// TwinCAT 3 PLC project EngineeringToolbox
// Title: EngineeringToolbox
// Company: Beckhoff Electronics Mfg
// Author: Daniel Schlingmann
// ProjectVersion: 3.1.2.2
// Description: Engineering Toolbox Library The library is provided "as-is" for TwinCAT3.1 by the Beckhoff Industry Management for Electronics Manufacturing. Please check the function "DisclaimerStatement : WSTRING[1500]" in additon to the following disclaimer: THE SOFTWARE IS PROVIDED "AS IS", WITHOUT WARRANTY OF ANY KIND, EXPRESS OR IMPLIED, INCLUDING BUT NOT LIMITED TO THE WARRANTIES OF MERCHANTABILITY, FITNESS FOR A PARTICULAR PURPOSE AND NONINFRINGEMENT. IN NO EVENT SHALL THE AUTHORS OR COPYRIGHT HOLDERS BE LIABLE FOR ANY CLAIM, DAMAGES OR OTHER LIABILITY, WHETHER IN AN ACTION OF CONTRACT, TORT OR OTHERWISE, ARISING FROM, OUT OF OR IN CONNECTION WITH THE SOFTWARE OR THE USE OR OTHER DEALINGS IN THE SOFTWARE.
// ProgramVersion: 3.1.4022.7
// libraries:
//   Tc2_Drive, * (Beckhoff Automation GmbH)
//   Tc2_EtherCAT, * (Beckhoff Automation GmbH)
//   Tc2_IoFunctions, * (Beckhoff Automation GmbH)
//   Tc2_Math, * (Beckhoff Automation GmbH)
//   Tc2_MC2, * (Beckhoff Automation GmbH)
//   Tc2_MC2_Camming, * (Beckhoff Automation GmbH)
//   Tc2_MC2_Drive, * (Beckhoff Automation GmbH)
//   Tc2_MC2_FlyingSaw, * (Beckhoff Automation GmbH)
//   Tc2_MDP, * (Beckhoff Automation GmbH)
//   Tc2_ModbusRTU, * (Beckhoff Automation GmbH)
//   Tc2_ModbusSrv, * (Beckhoff Automation GmbH)
//   Tc2_NC, * (Beckhoff Automation GmbH)
//   Tc2_NCI, * (Beckhoff Automation GmbH)
//   Tc2_NcKinematicTransformation, * (Beckhoff Automation GmbH)
//   Tc2_PlcInterpolation, * (Beckhoff Automation GmbH)
//   Tc2_SerialCom, * (Beckhoff Automation GmbH)
//   Tc2_Smtp, * (Beckhoff Automation GmbH)
//   Tc2_Standard, * (Beckhoff Automation GmbH)
//   Tc2_SUPS, * (Beckhoff Automation GmbH)
//   Tc2_System, * (Beckhoff Automation GmbH)
//   Tc2_TcpIp, * (Beckhoff Automation GmbH)
//   Tc2_Utilities, * (Beckhoff Automation GmbH)
//   Tc2_XmlDataSrv, * (Beckhoff Automation GmbH)
//   Tc3_Module, * (Beckhoff Automation GmbH)
//   Tc2_BackupRestoreEL6900,newest,Beckhoff Automation GmbH
// project tree:
//   GVLs/ Gvl.TcGVL (not stored), PARAM.TcGVL (not stored)
//   POUs/BoundsCheck/ boundsError.TcPOU (not stored), boundsOK.TcPOU (not stored), checkBounds.TcPOU (not stored), CheckBoundsInfo.TcPOU (not stored)
//   POUs/Connectivity/ADS/ AdsDataExchange.TcPOU (not stored)
//   POUs/Connectivity/ Ipv4Addr_TO_UDINT.TcPOU (not stored), U_DEVICE_COM_CACHE.TcDUT, U_IPv4Addr.TcDUT (not stored), isValidIPv4Addr.TcPOU (not stored)
//   POUs/Connectivity/TF6310-TcpServer/DeviceCom/ TCPDeviceCom_SendRecBytes.TcPOU (not stored), TCPDeviceCom_SendRecString.TcPOU (not stored)
//   POUs/Connectivity/TF6340-SerialCom/ComPortDeviceCom/ ComPortDeviceCom_BufferHandle.TcPOU (not stored), ComPortDeviceCom_SendRecBytes.TcPOU (not stored), ComPortDeviceCom_SendRecString.TcPOU (not stored), ComPortEL6x22BEasyConnect.TcPOU (not stored)
//   POUs/Connectivity/TF6340-SerialCom/ComPortBasic/ ComPortBackground.TcPOU (not stored), ComPortSendRec.TcPOU (not stored)
//   POUs/Connectivity/TF625x-Modbus/Master/TF6250-ModbusTcpServer/TCP/ ModbusTcpMaster.TcPOU (not stored)
//   POUs/Connectivity/TF625x-Modbus/Master/TF6250-ModbusTcpServer/UDP/ ModbusUdpMaster.TcPOU (not stored)
//   POUs/Connectivity/TF625x-Modbus/Master/TF6255-ModbusRtu/ ModbusRtuMaster22B.TcPOU (not stored), ModbusRtuMaster5B.TcPOU (not stored), ModbusRtuMasterPC.TcPOU (not stored)
//   POUs/Connectivity/TF625x-Modbus/Master/_Components/ ModbusJob.TcPOU (not stored), ModbusSlaveCom.TcPOU (not stored)
//   POUs/Connectivity/TF625x-Modbus/Slave/ ModbusSlaveBase.TcPOU
//   POUs/Connectivity/TF6310-TcpServer/TcpBasic/ TCPSendRecCtrl.TcPOU (not stored), TCPConnectionCtrl.TcPOU (not stored), TCPSocketCtrl.TcPOU (not stored)
//   POUs/Connectivity/TF6310-TcpServer/UdpBasic/ UDPSendRecCtrl.TcPOU (not stored), UDPServerCtrl.TcPOU (not stored), UDPSocketCtrl.TcPOU (not stored)
//   POUs/ControllerTools/ AverageFilter.TcPOU, PIDController.TcPOU (not stored), PT1Filter.TcPOU (not stored), signum.TcPOU (not stored), SlewRateLimitter.TcPOU (not stored), SlidingAverageExt.TcPOU (not stored), SlidingAverage.TcPOU (not stored), ThreePointController.TcPOU (not stored)
//   POUs/DataBuffer/ DoubleBuffer.TcPOU (not stored), Quicksort.TcPOU (not stored)
//   POUs/DataBuffer/Fifo/ Fifo.TcPOU (not stored), FifoExt.TcPOU (not stored), FifoLRealSimple.TcPOU (not stored), FifoBase.TcPOU (not stored)
//   POUs/DataBuffer/Ringbuffer/ RingbufferBase.TcPOU (not stored), Ringbuffer.TcPOU (not stored), RingbufferCharSimple.TcPOU (not stored), RingbufferExt.TcPOU (not stored), RingbufferByteSimple.TcPOU (not stored), RingbufferLRealSimple.TcPOU (not stored)
//   POUs/EventLogger/ EventsWriteToLogbook.TcPOU (not stored), EVENT_HANDLING_CONFIG.TcDUT (not stored), getEventClassPriority.TcPOU (not stored), getEventClassText.TcPOU, SOURCE_ID.TcDUT (not stored)
//   POUs/EventLogger/ReadEvents/ EventlogRead.TcPOU (not stored), EVENTLOG_READ_DATA.TcDUT (not stored), EVENTLOG_READ_HANDLEINFO.TcDUT (not stored), EVENTLOG_READ_STREAM.TcDUT (not stored), EVENTLOG_READ_STREAM_DATA_RAW.TcDUT, EVENTLOG_READ_STREAM_DATA_RAW_EX.TcDUT (not stored)
//   POUs/EventLogger/TriggerEvents/ EventHandling.TcPOU (not stored), EventHandlingGrp10.TcPOU (not stored), EventHandlingGrp25.TcPOU (not stored), EventHandlingGrp50.TcPOU (not stored), EventHandlingGrpCustomized.TcPOU, EventHandlingConfirmIsReq.TcPOU, EventHandlingStatisticInfo.TcPOU (not stored)
//   POUs/Fieldbus/CANopen/ CANopenMasterDiag.TcPOU (not stored), CANopenMasterIO.TcPOU (not stored)
//   POUs/Fieldbus/EAP/ EAP_PUB_SUB_IO.TcPOU (not stored), EAP_DEVICE_IO.TcPOU (not stored), EAP_PUB_VAR.TcPOU (not stored), EAP_SUB_VAR.TcPOU (not stored)
//   POUs/Fieldbus/EtherCAT/ EcCoEReadNewestDiagMsg.TcPOU (not stored), EcDiagBase.TcPOU (not stored), EcDiagBase_wEvents.TcPOU (not stored)
//   POUs/Fieldbus/EtherCAT/_Components/ EcMasterIO.TcPOU (not stored), EcMasterSupervisor.TcPOU, EcSlavesDiag.TcPOU (not stored), EcSlaveSupervisor.TcPOU (not stored), EC_MASTER_DEVICE_STATE.TcDUT (not stored), EC_SLAVE_DIAG_INFO_DATA.TcDUT
//   POUs/Fieldbus/Profibus/ ProfibusMasterDiag.TcPOU (not stored), ProfibusMasterIO.TcPOU (not stored)
//   POUs/Fieldbus/Profinet/ ProfinetControllerIO.TcPOU, ProfinetControllerIO_wEvents.TcPOU (not stored), ProfinetDeviceIO.TcPOU (not stored)
//   POUs/FileHandling/Basic/ FileHandling.TcPOU (not stored), ReadDirSimple.TcPOU, ReadDirSimpleExt.TcPOU (not stored)
//   POUs/FileHandling/TF6421-XmlServer/ XmlReadWrite.TcPOU, XmlReadWriteWithBackupFile.TcPOU (not stored)
//   POUs/IO/Analog/ AnalogIn.TcPOU (not stored), AnalogIn32.TcPOU (not stored), AnalogInELMBase.TcPOU (not stored), AnalogInELMSingleSampleDINT.TcPOU (not stored), AnalogInELMSingleSampleREAL.TcPOU (not stored), AnalogInREAL.TcPOU (not stored), AnalogOut.TcPOU (not stored)
//   POUs/IO/ BlowOffSensors.TcPOU, Button.TcPOU (not stored), ButtonExt.TcPOU (not stored), Fuse.TcPOU (not stored), InOut.TcPOU (not stored), InOutExt.TcPOU (not stored), Input.TcPOU (not stored), Output.TcPOU
//   POUs/IO/Cylinder/ Cylinder.TcPOU (not stored), CylinderExt.TcPOU, CylinderType4.TcPOU (not stored), I_Cylinder.TcIO (not stored)
//   POUs/IO/Drives/ AxDriveBase.TcPOU, AxDriveGetRef.TcPOU (not stored), I_AxDriveBase.TcIO (not stored)
//   POUs/IO/Drives/CoE/ AxDriveCoE.TcPOU (not stored), AxDriveCoE_wEvents.TcPOU (not stored), CiA_DS402Controlword.TcPOU, CiA_DS402Statusword.TcPOU (not stored), eCiA_DS402_CONTROL_CMD.TcDUT (not stored), eCiA_DS402_STATUS_STATE.TcDUT (not stored)
//   POUs/IO/Drives/CoE/EL72xx/ AxDriveCoE_EL72xxParam.TcPOU (not stored), CiA_DS402StatuswordEx7xxx.TcPOU (not stored)
//   POUs/IO/Drives/DC/Ey73xx/ AxDriveDC.TcPOU, AxDriveDC_wEvents.TcPOU (not stored)
//   POUs/IO/Drives/SoE/ AxDriveSoE_Ax5000CommutationCalib.TcPOU (not stored), AxDriveSoE_Ax5000CalcPower.TcPOU (not stored), AxDriveSoE_Ax5000SwitchParamSet.TcPOU (not stored), Ax580x.TcPOU (not stored), AxDriveSoE_Ax5000.TcPOU (not stored), AxDriveSoE_Ax5000Param.TcPOU (not stored), AxDriveSoE_Ax5000wEvents.TcPOU (not stored), AxDriveSoE_Rexroth.TcPOU
//   POUs/IO/Drives/SoE/Ax5000ParamSTRUCTs/P/ AX5000_P_0001.TcDUT (not stored), AX5000_P_0002.TcDUT (not stored), AX5000_P_0003.TcDUT (not stored), AX5000_P_0004.TcDUT (not stored), AX5000_P_0009.TcDUT (not stored), AX5000_P_0010.TcDUT (not stored), AX5000_P_0020.TcDUT (not stored), AX5000_P_0021.TcDUT (not stored), AX5000_P_0040.TcDUT (not stored), AX5000_P_0050.TcDUT (not stored), AX5000_P_0051.TcDUT (not stored), AX5000_P_0052.TcDUT, AX5000_P_0053.TcDUT (not stored), AX5000_P_0054.TcDUT (not stored), AX5000_P_0055.TcDUT (not stored), AX5000_P_0056.TcDUT (not stored), AX5000_P_0057.TcDUT (not stored), AX5000_P_0058.TcDUT (not stored), AX5000_P_0059.TcDUT (not stored), AX5000_P_0060.TcDUT (not stored), AX5000_P_0061.TcDUT (not stored), AX5000_P_0062.TcDUT (not stored), AX5000_P_0063.TcDUT (not stored), AX5000_P_0064.TcDUT (not stored), AX5000_P_0065.TcDUT (not stored), AX5000_P_0066.TcDUT (not stored), AX5000_P_0067.TcDUT (not stored), AX5000_P_0068.TcDUT (not stored), AX5000_P_0069.TcDUT (not stored), AX5000_P_0070.TcDUT (not stored), AX5000_P_0071.TcDUT (not stored), AX5000_P_0072.TcDUT (not stored), AX5000_P_0073.TcDUT, AX5000_P_0074.TcDUT (not stored), AX5000_P_0075.TcDUT (not stored), AX5000_P_0076.TcDUT (not stored), AX5000_P_0077.TcDUT (not stored), AX5000_P_0078.TcDUT (not stored), AX5000_P_0088.TcDUT (not stored), AX5000_P_0089.TcDUT (not stored), AX5000_P_0090.TcDUT (not stored), AX5000_P_0091.TcDUT (not stored), AX5000_P_0092.TcDUT, AX5000_P_0093.TcDUT (not stored), AX5000_P_0096.TcDUT (not stored), AX5000_P_0097.TcDUT (not stored), AX5000_P_0098_beckhoff.TcDUT (not stored), AX5000_P_0098_beckhoff_electrical_data.TcDUT (not stored), AX5000_P_0099.TcDUT (not stored), AX5000_P_0100.TcDUT (not stored), AX5000_P_0101.TcDUT (not stored), AX5000_P_0102.TcDUT (not stored), AX5000_P_0103.TcDUT (not stored), AX5000_P_0104.TcDUT (not stored), AX5000_P_0105.TcDUT (not stored), AX5000_P_0106.TcDUT (not stored), AX5000_P_0107.TcDUT (not stored), AX5000_P_0108.TcDUT (not stored), AX5000_P_0109.TcDUT (not stored), AX5000_P_0110.TcDUT (not stored), AX5000_P_0111.TcDUT (not stored), AX5000_P_0112.TcDUT (not stored), AX5000_P_0113.TcDUT (not stored), AX5000_P_0114.TcDUT (not stored), AX5000_P_0115.TcDUT (not stored), AX5000_P_0116.TcDUT (not stored), AX5000_P_0117.TcDUT (not stored), AX5000_P_0118.TcDUT (not stored), AX5000_P_0119.TcDUT (not stored), AX5000_P_0125.TcDUT (not stored), AX5000_P_0126.TcDUT, AX5000_P_0127.TcDUT (not stored), AX5000_P_0128.TcDUT, AX5000_P_0150.TcDUT, AX5000_P_0151.TcDUT (not stored), AX5000_P_0152.TcDUT (not stored), AX5000_P_0153.TcDUT (not stored), AX5000_P_0154.TcDUT (not stored), AX5000_P_0155.TcDUT (not stored), AX5000_P_0158.TcDUT (not stored), AX5000_P_0159.TcDUT (not stored), AX5000_P_0160.TcDUT, AX5000_P_0161.TcDUT (not stored), AX5000_P_0162.TcDUT (not stored), AX5000_P_0163.TcDUT, AX5000_P_0165.TcDUT (not stored), AX5000_P_0166.TcDUT (not stored), AX5000_P_0167.TcDUT (not stored), AX5000_P_0168.TcDUT (not stored), AX5000_P_0169.TcDUT (not stored), AX5000_P_0170.TcDUT (not stored), AX5000_P_0171.TcDUT (not stored), AX5000_P_0180.TcDUT, AX5000_P_0181.TcDUT (not stored), AX5000_P_0182.TcDUT (not stored), AX5000_P_0183.TcDUT, AX5000_P_0184.TcDUT (not stored), AX5000_P_0185.TcDUT (not stored), AX5000_P_0188.TcDUT (not stored), AX5000_P_0189.TcDUT (not stored), AX5000_P_0192.TcDUT (not stored), AX5000_P_0193.TcDUT (not stored), AX5000_P_0196.TcDUT (not stored), AX5000_P_0198.TcDUT (not stored), AX5000_P_0199.TcDUT (not stored), AX5000_P_0200.TcDUT (not stored), AX5000_P_0201.TcDUT, AX5000_P_0202.TcDUT (not stored), AX5000_P_0203.TcDUT (not stored), AX5000_P_0204.TcDUT (not stored), AX5000_P_0205.TcDUT (not stored), AX5000_P_0206.TcDUT (not stored), AX5000_P_0207.TcDUT (not stored), AX5000_P_0208.TcDUT (not stored), AX5000_P_0209.TcDUT (not stored), AX5000_P_0210.TcDUT, AX5000_P_0211.TcDUT (not stored), AX5000_P_0212.TcDUT (not stored), AX5000_P_0213.TcDUT (not stored), AX5000_P_0214.TcDUT, AX5000_P_0215.TcDUT (not stored), AX5000_P_0216.TcDUT (not stored), AX5000_P_0217.TcDUT (not stored), AX5000_P_0218.TcDUT (not stored), AX5000_P_0219.TcDUT (not stored), AX5000_P_0220.TcDUT (not stored), AX5000_P_0221.TcDUT (not stored), AX5000_P_0250.TcDUT (not stored), AX5000_P_0251.TcDUT (not stored), AX5000_P_0252.TcDUT (not stored), AX5000_P_0253.TcDUT (not stored), AX5000_P_0254.TcDUT (not stored), AX5000_P_0255.TcDUT (not stored), AX5000_P_0256.TcDUT (not stored), AX5000_P_0270.TcDUT, AX5000_P_0271.TcDUT (not stored), AX5000_P_0272.TcDUT (not stored), AX5000_P_0273.TcDUT (not stored), AX5000_P_0274.TcDUT, AX5000_P_0275.TcDUT (not stored), AX5000_P_0276.TcDUT, AX5000_P_0277.TcDUT (not stored), AX5000_P_0278.TcDUT (not stored), AX5000_P_0300.TcDUT (not stored), AX5000_P_0301.TcDUT (not stored), AX5000_P_0302.TcDUT (not stored), AX5000_P_0303.TcDUT (not stored), AX5000_P_0304.TcDUT (not stored), AX5000_P_0305.TcDUT (not stored), AX5000_P_0306.TcDUT (not stored), AX5000_P_0307.TcDUT (not stored), AX5000_P_0308.TcDUT (not stored), AX5000_P_0309.TcDUT (not stored), AX5000_P_0310.TcDUT (not stored), AX5000_P_0311.TcDUT, AX5000_P_0312.TcDUT (not stored), AX5000_P_0313.TcDUT, AX5000_P_0314.TcDUT (not stored), AX5000_P_0315.TcDUT (not stored), AX5000_P_0316.TcDUT (not stored), AX5000_P_0317.TcDUT (not stored), AX5000_P_0320.TcDUT (not stored), AX5000_P_0321.TcDUT (not stored), AX5000_P_0322.TcDUT (not stored), AX5000_P_0323.TcDUT (not stored), AX5000_P_0324.TcDUT, AX5000_P_0325.TcDUT, AX5000_P_0326.TcDUT (not stored), AX5000_P_0350.TcDUT (not stored), AX5000_P_0351.TcDUT (not stored), AX5000_P_0352.TcDUT (not stored), AX5000_P_0353.TcDUT (not stored), AX5000_P_0354.TcDUT (not stored), AX5000_P_0356.TcDUT (not stored), AX5000_P_0360.TcDUT (not stored), AX5000_P_0361.TcDUT (not stored), AX5000_P_0400.TcDUT (not stored), AX5000_P_0401.TcDUT (not stored), AX5000_P_0402.TcDUT (not stored), AX5000_P_0451.TcDUT (not stored), AX5000_P_0452.TcDUT (not stored), AX5000_P_0453.TcDUT (not stored), AX5000_P_0454.TcDUT (not stored), AX5000_P_0455.TcDUT (not stored), AX5000_P_0456.TcDUT, AX5000_P_0457.TcDUT (not stored), AX5000_P_0458.TcDUT (not stored), AX5000_P_0459.TcDUT (not stored), AX5000_P_0460.TcDUT (not stored), AX5000_P_0461.TcDUT (not stored), AX5000_P_0462.TcDUT (not stored), AX5000_P_0463.TcDUT (not stored), AX5000_P_0464.TcDUT (not stored), AX5000_P_0502.TcDUT (not stored), AX5000_P_0503.TcDUT (not stored), AX5000_P_0504.TcDUT (not stored), AX5000_P_0505.TcDUT (not stored), AX5000_P_0511.TcDUT (not stored), AX5000_P_0512.TcDUT (not stored), AX5000_P_0513.TcDUT (not stored), AX5000_P_0514.TcDUT (not stored), AX5000_P_0515.TcDUT (not stored), AX5000_P_0516.TcDUT (not stored), AX5000_P_0517.TcDUT (not stored), AX5000_P_0518.TcDUT (not stored), AX5000_P_0552.TcDUT (not stored), AX5000_P_0553.TcDUT (not stored), AX5000_P_0554.TcDUT (not stored), AX5000_P_0555.TcDUT (not stored), AX5000_P_0556.TcDUT, AX5000_P_0557.TcDUT (not stored), AX5000_P_0558.TcDUT (not stored), AX5000_P_0601.TcDUT (not stored), AX5000_P_0602.TcDUT, AX5000_P_0610.TcDUT, AX5000_P_0611.TcDUT (not stored), AX5000_P_0800.TcDUT (not stored), AX5000_P_0801.TcDUT (not stored), AX5000_P_0802.TcDUT (not stored), AX5000_P_0804.TcDUT, AX5000_P_0805.TcDUT (not stored), AX5000_P_0806.TcDUT (not stored), AX5000_P_0810.TcDUT (not stored), AX5000_P_0811.TcDUT (not stored), AX5000_P_0850.TcDUT (not stored), AX5000_P_0851.TcDUT (not stored), AX5000_P_0900.TcDUT (not stored), AX5000_P_0901.TcDUT (not stored), AX5000_P_0902.TcDUT (not stored), AX5000_P_0904.TcDUT (not stored), AX5000_P_0905.TcDUT, AX5000_P_0906.TcDUT (not stored), AX5000_P_0912.TcDUT (not stored), AX5000_P_1000.TcDUT, AX5000_P_1001.TcDUT (not stored), AX5000_P_1002.TcDUT (not stored), AX5000_P_1003.TcDUT (not stored), AX5000_P_1004.TcDUT, AX5000_P_1005.TcDUT (not stored), AX5000_P_1006.TcDUT (not stored), AX5000_P_1007.TcDUT (not stored), AX5000_P_1008.TcDUT (not stored), AX5000_P_1009.TcDUT (not stored), AX5000_P_1010.TcDUT (not stored), AX5000_P_1011.TcDUT (not stored), AX5000_P_1012.TcDUT (not stored), AX5000_P_1020.TcDUT (not stored), AX5000_P_1021.TcDUT (not stored), AX5000_P_1022.TcDUT (not stored), AX5000_P_2000.TcDUT (not stored), AX5000_P_2001.TcDUT (not stored), AX5000_P_2002.TcDUT (not stored)
//   POUs/IO/Drives/SoE/Ax5000ParamSTRUCTs/S/ AX5000_S_0001.TcDUT (not stored), AX5000_S_0002.TcDUT (not stored), AX5000_S_0007.TcDUT, AX5000_S_0011.TcDUT (not stored), AX5000_S_0012.TcDUT (not stored), AX5000_S_0013.TcDUT (not stored), AX5000_S_0015.TcDUT (not stored), AX5000_S_0016.TcDUT (not stored), AX5000_S_0017.TcDUT (not stored), AX5000_S_0018.TcDUT (not stored), AX5000_S_0024.TcDUT (not stored), AX5000_S_0029.TcDUT (not stored), AX5000_S_0030.TcDUT (not stored), AX5000_S_0031.TcDUT (not stored), AX5000_S_0032.TcDUT (not stored), AX5000_S_0033.TcDUT (not stored), AX5000_S_0034.TcDUT (not stored), AX5000_S_0035.TcDUT (not stored), AX5000_S_0036.TcDUT (not stored), AX5000_S_0037.TcDUT (not stored), AX5000_S_0040.TcDUT (not stored), AX5000_S_0043.TcDUT (not stored), AX5000_S_0044.TcDUT (not stored), AX5000_S_0045.TcDUT (not stored), AX5000_S_0046.TcDUT (not stored), AX5000_S_0047.TcDUT (not stored), AX5000_S_0048.TcDUT (not stored), AX5000_S_0051.TcDUT, AX5000_S_0053.TcDUT (not stored), AX5000_S_0055.TcDUT (not stored), AX5000_S_0076.TcDUT, AX5000_S_0079.TcDUT (not stored), AX5000_S_0080.TcDUT (not stored), AX5000_S_0081.TcDUT (not stored), AX5000_S_0082.TcDUT (not stored), AX5000_S_0083.TcDUT (not stored), AX5000_S_0084.TcDUT (not stored), AX5000_S_0085.TcDUT (not stored), AX5000_S_0086.TcDUT (not stored), AX5000_S_0091.TcDUT (not stored), AX5000_S_0092.TcDUT (not stored), AX5000_S_0095.TcDUT (not stored), AX5000_S_0099.TcDUT (not stored), AX5000_S_0100.TcDUT (not stored), AX5000_S_0101.TcDUT, AX5000_S_0103.TcDUT (not stored), AX5000_S_0104.TcDUT (not stored), AX5000_S_0106.TcDUT (not stored), AX5000_S_0107.TcDUT (not stored), AX5000_S_0109.TcDUT, AX5000_S_0110.TcDUT, AX5000_S_0111.TcDUT (not stored), AX5000_S_0112.TcDUT (not stored), AX5000_S_0113.TcDUT (not stored), AX5000_S_0119.TcDUT (not stored), AX5000_S_0120.TcDUT, AX5000_S_0124.TcDUT (not stored), AX5000_S_0126.TcDUT (not stored), AX5000_S_0130.TcDUT (not stored), AX5000_S_0131.TcDUT (not stored), AX5000_S_0134.TcDUT (not stored), AX5000_S_0135.TcDUT, AX5000_S_0136.TcDUT, AX5000_S_0137.TcDUT, AX5000_S_0143.TcDUT (not stored), AX5000_S_0149.TcDUT (not stored), AX5000_S_0159.TcDUT (not stored), AX5000_S_0160.TcDUT (not stored), AX5000_S_0161.TcDUT (not stored), AX5000_S_0162.TcDUT (not stored), AX5000_S_0163.TcDUT (not stored), AX5000_S_0169.TcDUT (not stored), AX5000_S_0170.TcDUT (not stored), AX5000_S_0179.TcDUT (not stored), AX5000_S_0185.TcDUT (not stored), AX5000_S_0186.TcDUT (not stored), AX5000_S_0187.TcDUT (not stored), AX5000_S_0188.TcDUT (not stored), AX5000_S_0189.TcDUT (not stored), AX5000_S_0196.TcDUT (not stored), AX5000_S_0200.TcDUT (not stored), AX5000_S_0201.TcDUT, AX5000_S_0203.TcDUT (not stored), AX5000_S_0204.TcDUT (not stored), AX5000_S_0206.TcDUT (not stored), AX5000_S_0207.TcDUT (not stored), AX5000_S_0216.TcDUT (not stored), AX5000_S_0217.TcDUT (not stored), AX5000_S_0219.TcDUT (not stored), AX5000_S_0254.TcDUT (not stored), AX5000_S_0256.TcDUT (not stored), AX5000_S_0257.TcDUT (not stored), AX5000_S_0267.TcDUT (not stored), AX5000_S_0273.TcDUT (not stored), AX5000_S_0274.TcDUT (not stored), AX5000_S_0292.TcDUT (not stored), AX5000_S_0295.TcDUT (not stored), AX5000_S_0296.TcDUT, AX5000_S_0347.TcDUT (not stored), AX5000_S_0348.TcDUT (not stored), AX5000_S_0372.TcDUT (not stored), AX5000_S_0374.TcDUT, AX5000_S_0375.TcDUT (not stored), AX5000_S_0380.TcDUT (not stored), AX5000_S_0381.TcDUT (not stored), AX5000_S_0383.TcDUT (not stored), AX5000_S_0384.TcDUT (not stored), AX5000_S_0390.TcDUT, AX5000_S_0403.TcDUT (not stored), AX5000_S_0405.TcDUT (not stored), AX5000_S_0409.TcDUT, AX5000_S_0410.TcDUT (not stored), AX5000_S_0429.TcDUT (not stored), AX5000_S_0432.TcDUT (not stored), AX5000_S_0435.TcDUT (not stored), AX5000_S_0436.TcDUT (not stored)
//   POUs/IO/Drives/Stepper/ AxDriveStepper.TcPOU (not stored), AxDriveStepperParam.TcPOU, AxDriveStepper_wEvents.TcPOU (not stored)
//   POUs/IO/EL-EP/ AnalogOut_EL2535.TcPOU (not stored), EL1262_Base.TcPOU (not stored), EL3681.TcPOU (not stored), EL1904.TcPOU (not stored), EL69xx.TcPOU (not stored), EL3356.TcPOU (not stored), Eyx9xx.TcPOU (not stored), ZB8610.TcPOU (not stored)
//   POUs/IO/EL-EP/EL9x/ EL9501.TcPOU (not stored), EL9576.TcPOU, EL95xxPowerTerminal.TcPOU (not stored), ELSystemTerminal.TcPOU (not stored)
//   POUs/IO/_EcSlaveFWUpdater/ EcSlaveDevFWUpdater.TcPOU (not stored)
//   POUs/IO/_EcSlaveInfoDataIO/ EcSlaveInfoData.TcPOU (not stored), EcSlaveInfoDataExt.TcPOU (not stored), I_EcSlaveInfoData.TcIO (not stored)
//   POUs/IO/EL-EP/EL3403/ EL3403.TcPOU (not stored), EL3403Logic.TcPOU (not stored)
//   POUs/IO/EL-EP/EP92xxPwrBox/ EP9214.TcPOU (not stored), EP9214_CHANNEL.TcPOU (not stored), EP9224_0037.TcPOU (not stored), EP9224_0037_CHANNEL.TcPOU (not stored)
//   POUs/IO/FreqConv/EtherCAT/DS402/ EcFcDS402_ComBase.TcPOU
//   POUs/IO/FreqConv/ IOFcCom.TcPOU
//   POUs/IO/Motors/ IOMotor.TcPOU (not stored), IOMotor2Dir.TcPOU (not stored), IOMotorStarDelta.TcPOU (not stored)
//   POUs/IO/[underDev]/ Cylinder_wUnitItf.TcPOU (not stored)
//   POUs/IO/_ItfActuators/ I_ActuatorBase.TcIO (not stored), I_ActuatorEnableDisable.TcIO (not stored), I_ActuatorFwdRev.TcIO (not stored), I_ActuatorFwdBwd.TcIO (not stored), I_ActuatorLeftRight.TcIO (not stored), I_ActuatorOnOff.TcIO, I_ActuatorOpenClose.TcIO (not stored), I_ActuatorPosNeg.TcIO (not stored), I_ActuatorStartStop.TcIO (not stored), I_ActuatorUpDown.TcIO (not stored), I_ActuatorWorkBase.TcIO (not stored)
//   POUs/IpcDiag/MDP/InfoModuls/ MDP_CPU.TcPOU (not stored), MDP_Fan.TcPOU (not stored), MDP_Mainboard.TcPOU (not stored), MDP_RaidSimple.TcPOU (not stored), MDP_ReadModulList.TcPOU (not stored), MDP_SiliconDrives.TcPOU (not stored), MDP_UPS.TcPOU (not stored)
//   POUs/IpcDiag/MDP/ MDP_Info.TcPOU (not stored), MDP_IpcDiag.TcPOU (not stored), MDP_IpcDiag_wEvents.TcPOU (not stored)
//   POUs/IpcDiag/ UPSStatus.TcPOU (not stored)
//   POUs/Logging/ DataFileLogger.TcPOU (not stored), DataUdpLogger.TcPOU (not stored), I_LogbookSubscriber.TcIO (not stored), I_Logbook.TcIO (not stored), Logbook.TcPOU (not stored), LogbookData.TcDUT (not stored), LogbookPuplisher.TcPOU (not stored), LogbookSubEventLog.TcPOU, LogbookSubSendMail.TcPOU (not stored), adsLogError.TcPOU (not stored), adsLogHint.TcPOU (not stored), adsLogWarn.TcPOU (not stored), LogbookSubSysLog.TcPOU (not stored), LogbookSubWriteFile.TcPOU (not stored), Logbook_wEventClass.TcPOU (not stored), adsLogwTcEventClass.TcPOU (not stored)
//   POUs/Motion/TF50xx-NC/00_Base/ I_AxNcPTP.TcIO (not stored), AxFbBase.TcPOU (not stored), AxRWParaBase.TcPOU, I_AxNcBase.TcIO (not stored)
//   POUs/Motion/TF50xx-NC/02_Options/Parameter/ AxPara.TcPOU (not stored), AxParaCtrl.TcPOU (not stored)
//   POUs/Motion/TF50xx-NC/03_Utilities/ AxAutoWriteSoftLimit.TcPOU (not stored), CoordinateTransformation2D.TcPOU (not stored), AxCalcPosBias.TcPOU (not stored), AxResonanceAvoidance.TcPOU (not stored) (excluded from build), AxSoftSyncDistance.TcPOU, AxStatemodel.TcPOU (not stored), AxAutoFct.TcPOU (not stored), AX_JOB.TcPOU (not stored), getOvrVelo.TcPOU (not stored)
//   POUs/Motion/TF50xx-NC/ AxNcPTPwJobs.TcPOU (not stored), AxNcBaseExt.TcPOU (not stored), AxNcPtpGear.TcPOU (not stored), AxNcBase.TcPOU (not stored), AxNcPTP.TcPOU (not stored)
//   POUs/Motion/TF5100-NCI/ NciChannel_wEvents.TcPOU (not stored), NciChannel.TcPOU (not stored)
//   POUs/Motion/TF511x-KIN/03_DUTs/Positions/ KIN_POSITIONS.TcPOU (not stored), KIN_POSITIONS_ACS_DUT.TcDUT (not stored), KIN_POSITIONS_MCS_DUT.TcDUT (not stored), U_KIN_POSITIONS.TcDUT (not stored)
//   POUs/Motion/TF511x-KIN/03_DUTs/Trafo/ KIN_CALCTRAFO_AXPOS_PARAM.TcPOU (not stored), KIN_STATE_OBSERVER_OID_PARAM.TcPOU (not stored), KIN_STATICTRAFO_PARAM.TcPOU (not stored), KIN_TOOLTRAFO_PARAM.TcPOU (not stored), UCS.TcPOU (not stored)
//   POUs/Motion/ VALUE_3D.TcPOU (not stored), VALUE_3D_DUT.TcDUT (not stored), VALUE_6D.TcPOU, VALUE_6D_DUT.TcDUT (not stored)
//   POUs/Safety/Diag/ SafetyLogicAndIOTerminalDiag.TcPOU (not stored), SafetyIODeviceDiagRead.TcPOU (not stored), SafetyIODeviceDiag_wEvents.TcPOU (not stored), SafetyIOsDiag.TcPOU (not stored), SafetyLogicTerminalDiag.TcPOU (not stored), SafetyPlcTerminalDiag.TcPOU (not stored)
//   POUs/StringHelper/ cutStrNumberToSeperator.TcPOU (not stored), cutStrToSeperator2.TcPOU (not stored), replaceUmlauts.TcPOU (not stored), cutStrToSeperator.TcPOU, cutWStrToSeperator.TcPOU (not stored), DWORD_TO_BINSTR_EXT.TcPOU (not stored), DWORD_TO_HEXSTR_EXT.TcPOU, getCntCharInStr.TcPOU (not stored), getCntCharInWStr.TcPOU (not stored), isWStringNumeric.TcPOU (not stored), HEXSTR_TO_DWORD.TcPOU (not stored), HEXSTR_TO_LWORD.TcPOU (not stored), INSERT_EXT.TcPOU (not stored), LWORD_TO_BINSTR_EXT.TcPOU (not stored), LWORD_TO_HEXSTR_EXT.TcPOU (not stored), readStrToSeperator.TcPOU (not stored), replaceInString.TcPOU (not stored), getFilledString.TcPOU (not stored), isStringNumeric.TcPOU (not stored), readWStrToSeperator.TcPOU (not stored), replaceInWString.TcPOU (not stored), U_MAX_STRING.TcDUT (not stored), U_MAX_WSTRING.TcDUT (not stored), WINSERT_EXT.TcPOU (not stored)
//   POUs/System/ SystemInfo.TcPOU (not stored), SystemInfo64.TcPOU (not stored) (excluded from build), SystemPulses.TcPOU (not stored), TaskInfo.TcPOU (not stored)
//   POUs/TimeHelper/ PartsPerTime.TcPOU (not stored), createTOD.TcPOU (not stored), getDateAndTimeDelta.TcPOU (not stored), getTonCountdown.TcPOU (not stored), LivebitCheck.TcPOU (not stored), Ontime.TcPOU (not stored), OntimeExt.TcPOU (not stored), OntimeSimple.TcPOU (not stored), Pulse.TcPOU, SensorTimeoutCheck.TcPOU (not stored), systemtimeInCam.TcPOU (not stored), systemtimeCmp.TcPOU (not stored), systemtimeInWin.TcPOU (not stored), TimeSwitch.TcPOU (not stored), TONRecord.TcPOU (not stored), TONTOF.TcPOU (not stored), VeloLinearMeasurement.TcPOU (not stored)
//   POUs/_Miscellaneous/64BitFunctions/ CLEARBIT64.TcPOU (not stored), CSETBIT64.TcPOU (not stored), GETBIT64.TcPOU (not stored), SETBIT64.TcPOU (not stored)
//   POUs/_Miscellaneous/ nextIdx.TcPOU (not stored), TC_VN_COLORS.TcDUT (not stored) (excluded from build), FbBase.TcPOU (not stored), CAM.TcPOU, CAM3D.TcPOU (not stored), COLOR.TcDUT (not stored), ERROR_HDL.TcPOU (not stored), FbBaseExt.TcPOU (not stored), FbBaseOutputs.TcPOU (not stored), getNoOfBits.TcPOU, LCID.TcDUT (not stored), eLCID.TcDUT (not stored), LOGx.TcPOU (not stored), OEECalculation.TcPOU (not stored), polynomial.TcPOU (not stored), RF_TRIG.TcPOU (not stored), scale.TcPOU (not stored), SEQUENCE_HDL.TcPOU (not stored), setNoOfBits.TcPOU, TEST_FB.TcPOU (not stored), TOGGLE.TcPOU (not stored), U_32BIT_DATATYPE.TcDUT (not stored), U_64BIT_DATATYPE.TcDUT (not stored), WIN.TcPOU (not stored)
//   POUs/_Miscellaneous/Conversions/ ADSERROR_TO_HRESULT.TcPOU (not stored), DWORD_TO_REAL_EX.TcPOU (not stored), HRESULT_TO_ADSERROR.TcPOU (not stored), REAL_TO_FMLREAL.TcPOU (not stored), LWORD_TO_LREAL_EX.TcPOU (not stored), SWAP_BYTES_OF_WORDS.TcPOU (not stored), SWAP_WORDS_OF_DWORD.TcPOU (not stored), SWAP_WORDS_OF_LWORD.TcPOU (not stored), ADSERROR_TO_WIN32ERROR.TcPOU, ADSERROR_TO_WSERROR.TcPOU (not stored), C_TO_F.TcPOU (not stored), DEGREES_TO_RPM.TcPOU (not stored), F_TO_C.TcPOU (not stored), GF_TO_N.TcPOU (not stored), TO_FMLREAL.TcPOU (not stored), MMIN_TO_MMS.TcPOU, MMS_TO_MMIN.TcPOU, N_TO_GF.TcPOU (not stored), RPM_TO_DEGREES.TcPOU (not stored)
//   POUs/Safety/ SafetyCircuit.TcPOU (not stored), SafetyGroupIO.TcPOU (not stored), SafetyPlcBackupRestore.TcPOU (not stored), SAFETY_CIRCUIT_STATUS.TcDUT (not stored)
//   POUs/Statemodel/control/ I_StatemodelBase.TcIO (not stored), I_Statemodel.TcIO, Statemodel.TcPOU (not stored)
//   POUs/Statemodel/ eMODE.TcDUT, eSTATE.TcDUT (not stored)
//   POUs/Statemodel/UnitTemplate/ I_Statemodel_Unit.TcIO (not stored), Statemodel_Unit.TcPOU (not stored)
//   POUs/Motion/TF50xx-NC/01_Main/ AxAdmin.TcPOU (not stored), AxHoming.TcPOU, AxMotion.TcPOU (not stored)
//   POUs/Motion/TF50xx-NC/02_Options/Motion/ AxSuperposition.TcPOU (not stored), AxMoveSinus.TcPOU (not stored), AxHomingOnBlock.TcPOU (not stored)
//   POUs/Motion/TF5100-NCI/01_Main/ NciAdmin.TcPOU (not stored), NciGrp.TcPOU (not stored), NciItp.TcPOU (not stored), NciMotion.TcPOU (not stored), NCI_REF.TcPOU (not stored)
//   POUs/Motion/TF5100-NCI/02_Options/Error/ NciChnEventHandling.TcPOU (not stored), NciEventHandling.TcPOU (not stored)
//   POUs/Motion/TF5100-NCI/02_Options/MFunctions/ NciMFnc.TcPOU (not stored)
//   POUs/Motion/TF5100-NCI/02_Options/PlcItp/ NciCreateItpTable.TcPOU (not stored), NciCreateItpTableEntryTemplate.TcPOU (not stored)
//   POUs/Motion/TF5100-NCI/02_Options/RParameter/ NCiReadWriteRParam.TcPOU (not stored)
//   POUs/Motion/TF511x-KIN/01_Main/ KinAdmin.TcPOU (not stored), KIN_REF.TcPOU (not stored)
//   POUs/Motion/TF511x-KIN/02_Options/ KinLockUnlockTrafoParam.TcPOU (not stored), KinWriteToolTrafoParam.TcPOU (not stored), KinWriteUCSTrafoParam.TcPOU (not stored)
//   POUs/Motion/TF511x-KIN/ KinChannel.TcPOU (not stored)
//   POUs/Motion/TF50xx-NC/02_Options/Coupling/ AxCamming.TcPOU (not stored), AxFlyingSaw.TcPOU (not stored), AxGear.TcPOU (not stored)
//   POUs/Motion/TF50xx-NC/02_Options/Error/ AxNcEventHandling.TcPOU (not stored), AxEventHandling.TcPOU (not stored)
//   POUs/Motion/TF50xx-NC/02_Options/Phasing/ AxPhasing.TcPOU (not stored)
//   POUs/Motion/TF50xx-NC/02_Options/TouchProbe/ AxTouchProbe.TcPOU (not stored)
//   POUs/StringHelper/ExtendedString/ ExtString.TcPOU (not stored), ExtWString.TcPOU (not stored), T_EXT_STRING.TcDUT (not stored), T_EXT_WSTRING.TcDUT (not stored)
//   POUs/TimeHelper/Conversions/ FILETIME_TO_DATE.TcPOU (not stored), LREAL_TO_TIME_SEC.TcPOU (not stored), FILETIME_TO_TOD.TcPOU (not stored), SYSTEMTIME_TO_TIME.TcPOU (not stored), SYSTEMTIME_TO_TIME_EX.TcPOU, SYSTEMTIME_TO_TOD.TcPOU (not stored), SYSTEMTIME_TO_DATE.TcPOU (not stored), TIME_TO_FMRLREAL.TcPOU, TIME_TO_SYSTEMTIME.TcPOU (not stored)
//   Version/ disclaimerStatement.TcPOU (not stored), Global_Version.TcGVL

// ---- POUs/Connectivity/U_DEVICE_COM_CACHE.TcDUT
TYPE U_DEVICE_COM_CACHE :
UNION
	Text				:	STRING(PARAM.DEVICE_COM_MAX_CACHE-1);
	Bytes				:	ARRAY[PARAM.DEVICE_COM_MIN_CACHE..PARAM.DEVICE_COM_MAX_CACHE] OF BYTE;	
END_UNION
END_TYPE

// ---- POUs/EventLogger/ReadEvents/EVENTLOG_READ_STREAM_DATA_RAW.TcDUT
TYPE EVENTLOG_READ_STREAM_DATA_RAW :
STRUCT
	cb						: DWORD;	
	InvokeId				: DWORD;	
	Id						: DWORD;
	SrcId					: DWORD;
	AdsAddr					: ARRAY [0..5] OF BYTE;
	AddrHint				: ARRAY [0..1] OF BYTE;
	Class					: DWORD;
	Flags					: DWORD;
	Prio					: DWORD;
	State					: DWORD;
	UserData				: DWORD;
	zFmtProgId				: STRING(31);

	TimeSignaled			: T_FILETIME; //In UTC
	TimeReseted				: T_FILETIME; //In UTC
	TimeConfirmed			: T_FILETIME; //In UTC

	evtData					: EVENTLOG_READ_STREAM_DATA_RAW_EX;
	
END_STRUCT
END_TYPE

// ---- POUs/Fieldbus/EtherCAT/_Components/EC_SLAVE_DIAG_INFO_DATA.TcDUT
TYPE EC_SLAVE_DIAG_INFO_DATA :
STRUCT
	Addr									:	WORD; //Slaves own physical address e.g. 1004 
	ConfigType								:	STRING(18); //Configured type e.g. EL1008 or EL7211 
	ConfigName								:	STRING(31); //Name as configured in IO-tree (type removed)
	ConfigTypeIdentity						:	STRING(18); //Configured type according identity e.g. AX5206-0000-0210
	ScannedTypeIdentity						:	STRING(18); //Scanned type according identitiy e.g. EL7201-9014
	
//	{attribute 'displaymode':='hex'}  	
//	DevType									:	DWORD; //EtherCAT device type of a slave
	{attribute 'displaymode':='hex'}  
	DevState								:	BYTE; //Device state constant e.g. 16#08=Tc2_EtherCAT.EC_DEVICE_STATE_OP
	DevStateText							:	STRING(60); //e.g. OP, INIT etc...
	DevStateBits							:	ST_EcSlaveStateBitsEx; //The structure contains bits showing the EtherCAT status (e.g. OP) and the link status )e.g. (EC_LINK_STATE_MISSING_LINK)

	{attribute 'displaymode':='hex'}  
	LinkState								:	BYTE; //Link state constant e.g. 0=Tc2_EtherCAT.EC_LINK_STATE_NOT_PRESENT
	{attribute 'displaymode':='bin'}  
	DataLinkStatusReg						:	WORD; //Data link status register status based on Topology of an EtherCAT slave from ESC register 0110/0111hex or 272/273dec. Status 0 is displayed if the slave cannot be reached or is offline	

	//Error information	
	CntOfCRCErrors							:	UDINT; //Total number of CRC-Errors on all four ports of the slave 
	NoOfAbnormalStateChanges				:	UDINT; //Shows how many times the slave status changed from available to INIT_NO_COMM e.g. unpluged
	
	//Topology information
	HotConnectNodeStart						:	BOOL; //Indicates that slaves is teh start of a hot-connect group (bit.3 of topology status)
	HotConnectSlave							:	BOOL; //Indicates that the slave is a part of a hot-connect group (bit.4 of topology status)
   	HCSlaveCountCfg  						:  UINT; //Shows number of attached slaves at HC node start
 	HCSlaveCountAct  						:  UINT; //Shows number of active slaves at HC node start
	{attribute 'displaymode':='bin'}  
	TopologyStatus					      	:  DWORD; (* Bits.0 = TRUE: Distributed clocks are supported
														 Bits.1 = TRUE: Distributed clocks are supported (64 bit)
														 Bits.2 = TRUE: Slave is present
														 Bits.3 = TRUE: Slave is start node of a Hot Connect group
														 Bits.4 = TRUE: Slave is in a Hot Connect group
														 Bits.5 = TRUE: Hot-connect is invalid at port B
														 Bits.6 = TRUE: Hot-connect is invalid at port C
														 Bits.7 = TRUE: Hot-connect is invalid at port D *)

   	TopoOwnPhysicalAddr  					:  UINT; //Can be different to "Addr" automatically assigned
   	AutoIncAddr   							:  UINT; //Dedicated auto-increment address of slave
   	PhysicalPortAddr    					:  ST_PortAddr; //Structure with phy. addr. information at port A…D
   	AutoIncPortAddr    				 		:  ST_PortAddr; //Structure with Auto inc. addr. information at port A…D
	ConfigIdentity							:	ST_EcSlaveIdentity; //EtherCAT identity data of an EtherCAT slave device, vendor Id, product code etc...
	ScannedIdentity							:	ST_EcSlaveIdentity; //EtherCAT identity data of an EtherCAT slave device, vendor Id, product code etc...
	
	ScannedSeq								:	UINT; //Logical/scanned sequence which can be different to configured seq. if hot-connect groups are used 
	{attribute 'displaymode':='bin'}   
	ErrorIdentCode							:	WORD; //Interal error identefier (Not in OP, CRC error increased, etc...
END_STRUCT
END_TYPE

// ---- POUs/IO/Drives/SoE/Ax5000ParamSTRUCTs/P/AX5000_P_0052.TcDUT
TYPE AX5000_P_0052 :
STRUCT
	Time_limitation_for_peak_current:UINT;
END_STRUCT
END_TYPE

// ---- POUs/IO/Drives/SoE/Ax5000ParamSTRUCTs/P/AX5000_P_0073.TcDUT
TYPE AX5000_P_0073 :
STRUCT
	Motor_peak_torque:UDINT;
END_STRUCT
END_TYPE

// ---- POUs/IO/Drives/SoE/Ax5000ParamSTRUCTs/P/AX5000_P_0092.TcDUT
TYPE AX5000_P_0092 :
STRUCT
	Configured_channel_peak_current:UDINT;
END_STRUCT
END_TYPE

// ---- POUs/IO/Drives/SoE/Ax5000ParamSTRUCTs/P/AX5000_P_0126.TcDUT
TYPE AX5000_P_0126 :
STRUCT
	Motor_continouse_stall_force:UDINT;
END_STRUCT
END_TYPE

// ---- POUs/IO/Drives/SoE/Ax5000ParamSTRUCTs/P/AX5000_P_0128.TcDUT
TYPE AX5000_P_0128 :
STRUCT
	Motor_peak_force:UDINT;
END_STRUCT
END_TYPE

// ---- POUs/IO/Drives/SoE/Ax5000ParamSTRUCTs/P/AX5000_P_0150.TcDUT
TYPE AX5000_P_0150 EXTENDS ST_AX5000_P_0150 :
STRUCT
(*
	Actual_lenght:UINT:=224;
	Max_lenght:UINT:=224;

	Manufacturer:UINT:=2;
	Feedback_type:UINT:=1;
	Feedback_type_string:STRING(29):='hallo';
	Feedback_use:UINT:=3;
	Feedback_direction:UINT:=1;
//{attribute 'hide'}
	Rsvd1:ARRAY[0..2] OF UINT;

	(*Powersettlings*)
	Control_voltage:UINT;
	Wait_time_after_power_up:UINT;
	Connector:UINT;
//	{attribute 'hide'}	
	Rsvd2:ARRAY[0..2] OF UINT;

	(*Process channel*)
		Process_interface:UINT;
		Conector2:UINT;
			(*rsvd*)
			// {attribute 'hide'}
				Rsvd3:ARRAY[0..1] OF UINT;
			(*Data*)
				(*Sin/Cos*)
					Resulution_per_rotation:UDINT;
					Length_per_signal_period:UDINT;
					Sin_gain_correction:UINT;
					Sin_offset_correction:UINT;
					Cos_gain_correction:UINT;
					Cos_offset_correction:UINT;
					Sin_Cos_1Vss_monitoring:UINT;
					// {attribute 'hide'}
					Rsvd4:ARRAY[0..10] OF UINT;
				(*TTL*)
					(*Resolution_per_rotation:UDINT;
					Length_per_signal_period:UDINT;
					rsvd5:ARRAY[0..15] OF UINT;*)
				(*Resolver*)
					(*Control_word:UINT;
					Number_of_poles:USINT;
					Exibition_frequency:USINT;
					Transformation_ratio:UINT;
					Phase_shift:UINT;
					Sin_cos_amplitude_monitoring:UINT;
						 {attribute 'hide'}
					rsvd6:UINT;
					Amplitude_monitoring_max_limit:UINT;
					Amplitude_monitoring_min_limit:UINT;
					Observer_bandwidth:UINT;
					Observer_correction_factor_Iq_to_acc:UINT;
						 {attribute 'hide'}
					rsvd7:ARRAY[0..4] OF UDINT;*)
				(*MES*)
					(*Control_word:UINT;
						 {attribute 'hide'}
					rsvd8:UINT;
					sin_offset:UINT;
					cos_offset:UINT;
					Sin_cos_Amplitude_correction:UINT;
						 {attribute 'hide'}
					rsvd9:UINT;
					Amplitude_monitoring_max_limit:UINT;
					Amplitude_monitoring_min_limit:UINT;
					Observer_bandwidth:UINT;
					Observer_correction_factor_Iq_to_acc:UINT;
						 {attribute 'hide'}
					rsvd10:ARRAY[0..4] OF UDINT;*)
				(*HTL*)
					(*Resulution_per_rotation:UDINT;
					Length_per_signal_period:UDINT;
						 {attribute 'hide'}
					rsvd11:ARRAY[0..15] OF UINT;*)
	(*Parameter channel*)
		Parameter_interface:UINT;
		Conector3:UINT;
		Identifier:UDINT;
		Bit_resolution_singelturn_position:UINT;
		Bit_resolution_multiturn_position:UINT;
		Number_of_clockcycles_to_get_singelturn_position:UINT;
		Number_of_clockcycles_to_get_multiturn_position:UINT;
		Digital_name_plate:UINT;
		commutation_mode_adjustable_commutation_offset:UINT;
		Linear_resolution_about_digital_interface_in_nm:UDINT;
		//	 {attribute 'hide'}
		Rsvd12:ARRAY[0..3] OF UINT;
		data:ARRAY[0..29] OF UINT;
	(*manufacturer limits settings*)
		Maximum_continous_operation_speed:UINT;
		Maximum_continous_mechenical_speed:UINT;
		Maximum_temperature:UINT;
		//	 {attribute 'hide'}
		Rsvd13:ARRAY[0..2] OF UINT;

	FeedbackOption :UDINT:=1;
	//	 {attribute 'hide'}
	Reserve :ARRAY[0..5] OF UINT;

*)
END_STRUCT
END_TYPE

// ---- POUs/IO/Drives/SoE/Ax5000ParamSTRUCTs/P/AX5000_P_0160.TcDUT
TYPE AX5000_P_0160 :
STRUCT
	Calibrate_commutation_offset:UINT;
END_STRUCT
END_TYPE

// ---- POUs/IO/Drives/SoE/Ax5000ParamSTRUCTs/P/AX5000_P_0163.TcDUT
TYPE AX5000_P_0163 :
STRUCT
	Scan_feedback1:UINT;
END_STRUCT
END_TYPE

// ---- POUs/IO/Drives/SoE/Ax5000ParamSTRUCTs/P/AX5000_P_0180.TcDUT
TYPE AX5000_P_0180 EXTENDS ST_AX5000_P_0180:
STRUCT
(*	Actual_lenght:UINT:=224;
	Max_lenght:UINT:=224;

	Manufacturer:UINT:=2;
	Feedback_type:UINT:=1;
	Feedback_type_string:STRING(29):='';
	Feedback_use:UINT:=3;
	Feedback_direction:UINT:=1;
	(*rsvd*)
//{attribute 'hide'}
		rsvd1:ARRAY[0..2] OF UINT;

	(*Powersettlings*)
		Control_voltage:UINT;
		Wait_time_after_power_up:UINT;
		Connector:UINT;
//	{attribute 'hide'}
		Rsvd2:ARRAY[0..2] OF UINT;

	(*Process channel*)
		Process_interface:UINT;
		Conector2:UINT;
			(*rsvd*)
		//	{attribute 'hide'}
				Rsvd3:ARRAY[0..1] OF UINT;
			(*Data*)
				(*Sin/Cos*)
					Resulution_per_rotation:UDINT;
					Length_per_signal_period:UDINT;
					Sin_gain_correction:UINT;
					Sin_offset_correction:UINT;
					Cos_gain_correction:UINT;
					Cos_offset_correction:UINT;
					Sin_Cos_1Vss_monitoring:UINT;
					Rsvd4:ARRAY[0..10] OF UINT;
				(*TTL*)
					(*Resolution_per_rotation:UDINT;
					Length_per_signal_period:UDINT;
				//	{attribute 'hide'}
					rsvd5:ARRAY[0..15] OF UINT;*)
				(*Resolver*)
					(*Control_word:UINT;
					Number_of_poles:USINT;
					Exibition_frequency:USINT;
					Transformation_ratio:UINT;
					Phase_shift:UINT;
					Sin_cos_amplitude_monitoring:UINT;
				//	{attribute 'hide'}
					rsvd6:UINT;
					Amplitude_monitoring_max_limit:UINT;
					Amplitude_monitoring_min_limit:UINT;
					Observer_bandwidth:UINT;
					Observer_correction_factor_Iq_to_acc:UINT;
					rsvd7:ARRAY[0..4] OF UDINT;*)
				(*MES*)
					(*Control_word:UINT;
				//	{attribute 'hide'}
					rsvd8:UINT;
					sin_offset:UINT;
					cos_offset:UINT;
					Sin_cos_Amplitude_correction:UINT;
					rsvd9:UINT;
					Amplitude_monitoring_max_limit:UINT;
					Amplitude_monitoring_min_limit:UINT;
					Observer_bandwidth:UINT;
					Observer_correction_factor_Iq_to_acc:UINT;
				//	{attribute 'hide'}
					rsvd10:ARRAY[0..4] OF UDINT;*)
				(*HTL*)
					(*Resulution_per_rotation:UDINT;
					Length_per_signal_period:UDINT;
					rsvd11:ARRAY[0..15] OF UINT;*)
	(*Parameter channel*)
		Parameter_interface:UINT;
		Conector3:UINT;
		Identifier:UDINT;
		Bit_resolution_singelturn_position:UINT;
		Bit_resolution_multiturn_position:UINT;
		Number_of_clockcycles_to_get_singelturn_position:UINT;
		Number_of_clockcycles_to_get_multiturn_position:UINT;
		Digital_name_plate:UINT;
		commutation_mode_adjustable_commutation_offset:UINT;
		Linear_reselution_about_digital_interface_in_nm:UDINT;
	//	{attribute 'hide'}
		Rsvd12:ARRAY[0..3] OF UINT;
		Data:ARRAY[0..29] OF UINT;
	(*manufacturer limits settings*)
		Maximum_continous_operation_speed:UINT;
		Maximum_continous_mechenical_speed:UINT;
		Maximum_temperature:UINT;
	//	{attribute 'hide'}
		Rsvd13:ARRAY[0..2] OF UINT;

	FeedbackOption :UDINT:=1;
//	{attribute 'hide'}
	Rsvd14 :ARRAY[0..5] OF UINT;
*)
END_STRUCT
END_TYPE

// ---- POUs/IO/Drives/SoE/Ax5000ParamSTRUCTs/P/AX5000_P_0183.TcDUT
TYPE AX5000_P_0183 :
STRUCT
	Feedback_2_geat_denominator:UDINT;
END_STRUCT
END_TYPE

// ---- POUs/IO/Drives/SoE/Ax5000ParamSTRUCTs/P/AX5000_P_0201.TcDUT
TYPE AX5000_P_0201 :
STRUCT
	Nominal_main_voltage:UINT;
END_STRUCT
END_TYPE

// ---- POUs/IO/Drives/SoE/Ax5000ParamSTRUCTs/P/AX5000_P_0210.TcDUT
TYPE AX5000_P_0210 :
STRUCT
	External_brak_resistor_actual_continouse_power:UINT;
END_STRUCT
END_TYPE

// ---- POUs/IO/Drives/SoE/Ax5000ParamSTRUCTs/P/AX5000_P_0214.TcDUT
TYPE AX5000_P_0214 :
STRUCT
	DC_Link_connection_mode:UINT;
END_STRUCT
END_TYPE

// ---- POUs/IO/Drives/SoE/Ax5000ParamSTRUCTs/P/AX5000_P_0270.TcDUT
{attribute 'pack_mode' := '1'}//Ensures 1-byte-alignmend
TYPE AX5000_P_0270 :
STRUCT
	Actual_lenght:UINT;
	Max_lenght:UINT;
	Feedback1:STRING(29);
//	{attribute 'hide'}
	Rsvd1:UINT;
	Serial_number_feedback1:ARRAY[0..1] OF UDINT;
	Feedback2:STRING(29);
//	{attribute 'hide'}
	Rsvd2:UINT;
	Serial_number_feedback2:ARRAY[0..1] OF UDINT;
	Modulo_value:UDINT;

(*Data read from file*)

(*data[0][0]*)
	Feedback_number1:UINT;
	Data_set1:UINT;
	Feedback_position1:UDINT;
	Modulo_position1:UDINT;
	Crc1:UDINT;
(*data[0][1]*)
	Feedback_number2:UINT;
	Data_se2t:UINT;
	Feedback_position2:UDINT;
	Modulo_position2:UDINT;
	Crc2:UDINT;
(*data[1][0]*)
	Feedback_number3:UINT;
	Data_set3:UINT;
	Feedback_position3:UDINT;
	Modulo_position3:UDINT;
	Crc3:UDINT;
(*data[1][1]*)
	Feedback_number4:UINT;
	Data_set4:UINT;
	Feedback_position4:UDINT;
	Modulo_position4:UDINT;
	Crc4:UDINT;


(*Current Data*)


(*data[0][0]*)
	Feedback_number5:UINT;
	Data_set5:UINT;
	Feedback_position5:UDINT;
	Modulo_position5:UDINT;
	Crc5:UDINT;
(*data[0][1]*)
	Feedback_number6:UINT;
	Data_se6t:UINT;
	Feedback_position6:UDINT;
	Modulo_position:UDINT;
	Crc6:UDINT;
(*data[1][0]*)
	Feedback_number7:UINT;
	Data_set7:UINT;
	Feedback_position7:UDINT;
	Modulo_position7:UDINT;
	Crc7:UDINT;
(*data[1][1]*)
	Feedback_number8:UINT;
	Data_set8:UINT;
	Feedback_position8:UDINT;
	Modulo_position8:UDINT;
	Crc8:UDINT;
END_STRUCT
END_TYPE

// ---- POUs/IO/Drives/SoE/Ax5000ParamSTRUCTs/P/AX5000_P_0274.TcDUT
{attribute 'pack_mode' := '1'}
TYPE AX5000_P_0274 :
STRUCT
	Actual_lenght:UINT;
	Max_lenght:UINT;
	Position_offset_feedback_1:UDINT;
	Position_offset_feedback_2:UDINT;
END_STRUCT
END_TYPE

// ---- POUs/IO/Drives/SoE/Ax5000ParamSTRUCTs/P/AX5000_P_0276.TcDUT
TYPE AX5000_P_0276 :
STRUCT
	Data_storage_feedback1_Data_storge_feedback2:UDINT;	(*Data_storage_feedback1 8Bit; Data_storage_feedback2 8 Bit*)
END_STRUCT
END_TYPE

// ---- POUs/IO/Drives/SoE/Ax5000ParamSTRUCTs/P/AX5000_P_0311.TcDUT
TYPE AX5000_P_0311 :
STRUCT
	PLL_ctrl_error:DINT;
END_STRUCT
END_TYPE

// ---- POUs/IO/Drives/SoE/Ax5000ParamSTRUCTs/P/AX5000_P_0313.TcDUT
TYPE AX5000_P_0313 :
STRUCT
	Actual_lenght:UINT;
	Max_lenght:UINT;
	String_output_mode:UINT;
	Backlight_mode:UINT;
	Keypad_mode:UINT;
//	{attribute 'hide'}
	Rsvd:UINT;
	Output_string:STRING(39);
END_STRUCT
END_TYPE

// ---- POUs/IO/Drives/SoE/Ax5000ParamSTRUCTs/P/AX5000_P_0324.TcDUT
TYPE AX5000_P_0324 :
STRUCT
	Actual_lenght:UINT;
	Max_lenght:UINT;
	ProductCode_RevisionNo:STRING;
END_STRUCT
END_TYPE

// ---- POUs/IO/Drives/SoE/Ax5000ParamSTRUCTs/P/AX5000_P_0325.TcDUT
TYPE AX5000_P_0325 :
STRUCT
	Actual_lenght:UINT;
	Max_lenght:UINT;
	Compile_time_and_date:STRING;
END_STRUCT
END_TYPE

// ---- POUs/IO/Drives/SoE/Ax5000ParamSTRUCTs/P/AX5000_P_0456.TcDUT
TYPE AX5000_P_0456 :
STRUCT
	Actual_motor_voltage_phase_U:UINT;
END_STRUCT
END_TYPE

// ---- POUs/IO/Drives/SoE/Ax5000ParamSTRUCTs/P/AX5000_P_0556.TcDUT
TYPE AX5000_P_0556 :
STRUCT
	Position_interpolator_type:UINT;
END_STRUCT
END_TYPE

// ---- POUs/IO/Drives/SoE/Ax5000ParamSTRUCTs/P/AX5000_P_0602.TcDUT
TYPE AX5000_P_0602 :
STRUCT
	Predictive_torque_command_value:INT;
END_STRUCT
END_TYPE

// ---- POUs/IO/Drives/SoE/Ax5000ParamSTRUCTs/P/AX5000_P_0610.TcDUT
{attribute 'pack_mode' := '1'}
TYPE AX5000_P_0610 :
STRUCT
	Actual_lenght:UINT;
	Max_lenght:UINT;
	Velocity_limit:DINT;
	Velocity_condition:UINT;
//	{attribute 'hide'}
	Rsvd:UINT;
	Torque_force_limit:UINT;
//	{attribute 'hide'}
	Rsvd1:UINT;
	Torque_force_condition:UINT;
//	{attribute 'hide'}
	Rsvd2:UINT;
//	{attribute 'hide'}
	Rsvd3:UDINT;
//	{attribute 'hide'}
	Rsvd4:UDINT;
END_STRUCT
END_TYPE

// ---- POUs/IO/Drives/SoE/Ax5000ParamSTRUCTs/P/AX5000_P_0804.TcDUT
TYPE AX5000_P_0804 :
STRUCT
	Digital_feedback_inputs_option_unit:UINT;
END_STRUCT
END_TYPE

// ---- POUs/IO/Drives/SoE/Ax5000ParamSTRUCTs/P/AX5000_P_0905.TcDUT
TYPE AX5000_P_0905 :
STRUCT
	Clear_error_history:UINT;
END_STRUCT
END_TYPE

// ---- POUs/IO/Drives/SoE/Ax5000ParamSTRUCTs/P/AX5000_P_1000.TcDUT
TYPE AX5000_P_1000 :
STRUCT
	Debug_pointer_1_adr:UDINT;
END_STRUCT
END_TYPE

// ---- POUs/IO/Drives/SoE/Ax5000ParamSTRUCTs/P/AX5000_P_1004.TcDUT
TYPE AX5000_P_1004 :
STRUCT
	Debug_pointer_2_type:UINT;
END_STRUCT
END_TYPE

// ---- POUs/IO/Drives/SoE/Ax5000ParamSTRUCTs/S/AX5000_S_0007.TcDUT
TYPE AX5000_S_0007 :
STRUCT
	Feedvack_acquisition_capture_point:UINT;
END_STRUCT
END_TYPE

// ---- POUs/IO/Drives/SoE/Ax5000ParamSTRUCTs/S/AX5000_S_0051.TcDUT
TYPE AX5000_S_0051 :
STRUCT
	Position_feedback_value_1:DINT;
END_STRUCT
END_TYPE

// ---- POUs/IO/Drives/SoE/Ax5000ParamSTRUCTs/S/AX5000_S_0076.TcDUT
TYPE AX5000_S_0076 EXTENDS ST_AX5000_S_0076:
STRUCT
//	Position_data_scaling_type:UINT;
END_STRUCT
END_TYPE

// ---- POUs/IO/Drives/SoE/Ax5000ParamSTRUCTs/S/AX5000_S_0101.TcDUT
TYPE AX5000_S_0101 :
STRUCT
	Velocity_loop_integral_action_time:UINT;
END_STRUCT
END_TYPE

// ---- POUs/IO/Drives/SoE/Ax5000ParamSTRUCTs/S/AX5000_S_0109.TcDUT
TYPE AX5000_S_0109 :
STRUCT
	Motor_peak_current:UDINT;
END_STRUCT
END_TYPE

// ---- POUs/IO/Drives/SoE/Ax5000ParamSTRUCTs/S/AX5000_S_0110.TcDUT
TYPE AX5000_S_0110 :
STRUCT
	Amplifier_peak_current:UDINT;
END_STRUCT
END_TYPE

// ---- POUs/IO/Drives/SoE/Ax5000ParamSTRUCTs/S/AX5000_S_0120.TcDUT
TYPE AX5000_S_0120 :
STRUCT
	Current_controler_loop_integral_action_time2:UINT;
END_STRUCT
END_TYPE

// ---- POUs/IO/Drives/SoE/Ax5000ParamSTRUCTs/S/AX5000_S_0135.TcDUT
TYPE AX5000_S_0135 :
STRUCT
	Drive_status_word:UINT;
END_STRUCT
END_TYPE

// ---- POUs/IO/Drives/SoE/Ax5000ParamSTRUCTs/S/AX5000_S_0136.TcDUT
TYPE AX5000_S_0136 :
STRUCT
	Positive_acceleration_limit_value:UDINT;
END_STRUCT
END_TYPE

// ---- POUs/IO/Drives/SoE/Ax5000ParamSTRUCTs/S/AX5000_S_0137.TcDUT
TYPE AX5000_S_0137 :
STRUCT
	Negative_acceleration_limit_value:UDINT;
END_STRUCT
END_TYPE

// ---- POUs/IO/Drives/SoE/Ax5000ParamSTRUCTs/S/AX5000_S_0201.TcDUT
TYPE AX5000_S_0201 :
STRUCT
	Motor_warning_temperature:UINT;
END_STRUCT
END_TYPE

// ---- POUs/IO/Drives/SoE/Ax5000ParamSTRUCTs/S/AX5000_S_0296.TcDUT
TYPE AX5000_S_0296 :
STRUCT
	Velocity_feed_forword_gain:UINT;
END_STRUCT
END_TYPE

// ---- POUs/IO/Drives/SoE/Ax5000ParamSTRUCTs/S/AX5000_S_0374.TcDUT
TYPE AX5000_S_0374 :
STRUCT
	Actual_lenght:UINT;
	Max_lenght:UINT;
	Procedure_command_error_list:ARRAY[0..59] OF UINT;
END_STRUCT
END_TYPE

// ---- POUs/IO/Drives/SoE/Ax5000ParamSTRUCTs/S/AX5000_S_0390.TcDUT
TYPE AX5000_S_0390 :
STRUCT
	Diagnostic_number:UDINT;
END_STRUCT
END_TYPE

// ---- POUs/IO/Drives/SoE/Ax5000ParamSTRUCTs/S/AX5000_S_0409.TcDUT
TYPE AX5000_S_0409 :
STRUCT
	Probe1_positive_latched:UINT;
END_STRUCT
END_TYPE

// ---- POUs/Statemodel/eMODE.TcDUT
{attribute 'qualified_only'}
//Default mode enum 0 - 10
{attribute 'to_string'}
TYPE eMODE :
(
	IDLE		 		:= 0,	
	MANUAL				:= 1,
	AUTO				:= 2,
	SEMI_AUTO			:= 3,
	SETUP				:= 4,
	STEP				:= 5,
	PRODUCTION			:= 6,
	MAINTENANCE			:= 7,
	SERVICE				:= 8,
	INIT				:= 9
				
);
END_TYPE

// ---- Version/Global_Version.TcGVL
{attribute 'TcGenerated'}
{attribute 'no-analysis'}
{attribute 'linkalways'}
// This function has been automatically generated from the project information.
VAR_GLOBAL CONSTANT
	{attribute 'const_non_replaced'}
	stLibVersion_EngineeringToolbox : ST_LibVersion := (iMajor := 3, iMinor := 1, iBuild := 2, iRevision := 2, nFlags := 1, sVersion := '3.1.2.2');
END_VAR

// ---- POUs/IO/_ItfActuators/I_ActuatorOnOff.TcIO
INTERFACE I_ActuatorOnOff EXTENDS I_ActuatorBase

{attribute 'monitoring' := 'call'}
PROPERTY public isOn : BOOL
GET
END_GET
END_PROPERTY

METHOD public switchOn : BOOL
VAR_INPUT
END_VAR
END_METHOD

END_INTERFACE

// ---- POUs/Statemodel/control/I_Statemodel.TcIO
INTERFACE I_Statemodel extends I_StatemodelBase

METHOD PUBLIC FINAL addSlave : BOOL
VAR_INPUT
	ipSlave					:	I_Statemodel;
END_VAR
END_METHOD

METHOD PUBLIC isModeActive : BOOL
VAR_INPUT
	Mode													: eMODE;				
END_VAR
END_METHOD

METHOD PUBLIC isStateActive : BOOL
VAR_INPUT
	state						:	eSTATE;
END_VAR
END_METHOD

PROPERTY public remoteData : U_64BIT_DATATYPE
GET
END_GET
SET
END_SET
END_PROPERTY

{attribute 'monitoring' := 'call'}
PROPERTY PUBLIC rErrHdl : REFERENCE to ERROR_HDL
GET
END_GET
END_PROPERTY

METHOD PUBLIC reset : boOL //Result = TRUE if Resetting finished - ErrHdl.Flag = FALSE
VAR_INPUT
END_VAR
END_METHOD

METHOD PUBLIC setLocalError : booL
VAR_INPUT
END_VAR
END_METHOD

END_INTERFACE

// ---- POUs/Connectivity/TF625x-Modbus/Slave/ModbusSlaveBase.TcPOU
{attribute 'no_check'}
// Modbus SlaveRoot 
// This Funktionblock represents a root structure for a Modbus slave to communicate with all Modbus masters of Engineering Toolbox 
// inherit this POU into "your" Modbus device POU
// declare "your" Data POU for your Modbus Device
// overload methodes evaluation, initJobs and prepareWriteData as private and edit inbetween the marks
// call methode Run to start communication.
// based on TF625x Modbus communication
FUNCTION_BLOCK ModbusSlaveBase      
VAR_INPUT
	IpAddr													:	T_IPv4Addr := '127.0.0.1';	// use only for TCP and UDP or ''
	Port 													:	UDINT;			// use only for TCP			or 0
	Address													:	BYTE := 0;		//Modbus RTU addres
//	Data													:	MyModbusDeviceData;	
END_VAR            							
VAR_OUTPUT
	ModBusCom												:	ModbusSlaveCom; //Master-Slave Handshake object
	Valid													:	BOOL; 		//	data valid 
	TimeStamp												:	DT;			//	timestamp of last refresh 
	CountGood												:	DWORD := 0;	//	counter for successful data transmission 
	CountBad												:	DWORD := 0;	//	counter for failed data transmission
	NoOfJobs												:	INT;		//	no of active jobs
END_VAR
VAR
(* memory **************************************************)
	state													:	INT;						
(* trigger *************************************************)

(* timer ***************************************************)

(* blocks **************************************************)

(* internal used variables *********************************)
	i,j,k													:	INT :=0;	
END_VAR

;

METHOD PROTECTED evaluation : BOOL //Result needs to be TRUE if data are evaluated
VAR_INPUT
	CurrentJobIdx						: INT;
END_VAR
// copy and edit the code only between the marks to evaluate read data
	
	CASE currentJobIdx OF
	0: evaluation											:= TRUE;
	// **********************************************************		
	// Modify start *********************************************	
	1:	// evaluation of job 1 
		// Data.Var_a										:= ModBusCom.Data[1];
		// MEMCPY(ADR(Data.Var_b), ADR(ModBusCom.Data[1]),SIZEOF(Data.Var_b));
			// HOST_TO_BE16(Data.Var_b);		
		// MEMCPY(ADR(Data.Var_c), ADR(ModBusCom.Data[2]),SIZEOF(Data.Var_c));
			// HOST_TO_BE32(Data.Var_c);				
		//evaluation										:= TRUE;
	2:	// evaluation of job 2 
		// MEMCPY(ADR(Data.Var_d), ADR(ModBusCom.Data[1]),SIZEOF(Data.Var_a));
		// Data.Var_e										:=	DWORD_TO_REAL_EX(	ADR(ModBusCom.Data[	5	]));
		// Data.Var_f										:=	DWORD_TO_REAL_EX(	ADR(ModBusCom.Data[	9	]));	
		//evaluation										:= TRUE;	                                                
	3: 	// evaluation of job 3                              
		// Data.Var_g										:=	TO_INT(					ModBusCom.Data[	1	]);	
		// Data.Var_h										:=	TO_INT(					ModBusCom.Data[	3	]);
		// Data.Var_i										:=	TO_INT(					ModBusCom.Data[	5	]);
		//evaluation										:= TRUE;																					
	4:	// write job, no evaluation 	
		//evaluation										:= TRUE;
	// Modify end ***********************************************
	// **********************************************************
	ELSE
		;
	END_CASE
END_METHOD

METHOD PROTECTED initJobs : BOOL //Result needs to be TRUE for every valid JobIdx 
VAR_INPUT
	JobIdx													:	INT;
END_VAR
(********** Modbus slave jobs *********************)
	
// HINT: The register number is in accordance with the Modbus specification always less 1.
	CASE JobIdx OF
	0:initJobs												:= TRUE;
// **********************************************************		
// Modify start *********************************************
	1: // read job 
//		ModBusCom.Jobs[JobIdx].FunctionCode 				:=   3		;
//		ModBusCom.Jobs[JobIdx].startAddress					:=   499	;	(* first read-address -1 *)
//		ModBusCom.Jobs[JobIdx].Quantity 					:=   14		;	(* no of read words *)
//		initJobs											:= TRUE;
		                                    				
	2:	// read job                         				
//		ModBusCom.Jobs[JobIdx].FunctionCode 				:=   3		;
//		ModBusCom.Jobs[JobIdx].startAddress					:=  40000	;	(* first read-address -1 *)
//		ModBusCom.Jobs[JobIdx].Quantity 					:=   120	;	(* no of read words *)
//		initJobs											:= TRUE;
	3:	// read job                         				
//		ModBusCom.Jobs[JobIdx].FunctionCode 				:=   3		;
//		ModBusCom.Jobs[JobIdx].startAddress					:=  40120	;	(* first read-address -1 *)
//		ModBusCom.Jobs[JobIdx].Quantity 					:=   20		;	(* no of read words *)
//		initJobs											:= TRUE;
	4:	// write job                        				
//		ModBusCom.Jobs[JobIdx].FunctionCode 				:=   5		;
//		ModBusCom.Jobs[JobIdx].startAddress					:=   112	;	(* first read-address*)
//		ModBusCom.Jobs[JobIdx].Quantity 					:=   1		;	(* no of write words *)
//		initJobs											:= TRUE;
// Modify end ***********************************************
// **********************************************************	

	ELSE	
		;
	END_CASE
END_METHOD

METHOD PROTECTED prepareWriteData : BOOL	//Result needs to be TRUE for every valid write JobIdx
VAR_INPUT
	CurrentJobIdx						: INT;
END_VAR
// copy and edit the code only between the marks to prepare necessary write data
	CASE currentJobIdx OF	
	0:prepareWriteData										:= TRUE;
	// **********************************************************		
	// Modify start *********************************************
	1:	// no write data in this job
		
	2:	// no write data in this job
											
	3:  // no write data in this job
	
	4:	//Copy write job data to com object
		// ModBusCom.Data[	1	]							:=	Data.SET_Var_j;
		// prepareWriteData									:= TRUE; //Set to true:              			
	// Modify end ***********************************************
	// **********************************************************		
	ELSE
		;
	END_CASE
END_METHOD

METHOD FINAL run : BOOL // returns TRUE if one job is finished
VAR_INPUT
	Enable													:	BOOL;
END_VAR
	(* Modbus slave logic 									*)
	(********************************************************)
	
(* Sequence ****************************************************************)
CASE state OF 
//Wait for start slave 
0: 
	IF Enable 
	THEN
		ModBusCom.Enable									:= Enable;
		ModBusCom.Address 									:= Address;
		ModBusCom.IpAddr	 								:= IpAddr;
		ModBusCom.Port	 									:= Port;
		ModBusCom.countBad 		:= ModBusCom.countGood		:= 0;
		ModBusCom.noOfJobs 									:= 0;
		
		//Run loop to init every single job		
		FOR i:= ModBusCom.MIN_SLAVE_JOB TO ModBusCom.MAX_SLAVE_JOB DO
			ModBusCom.Jobs[i].Init();
			IF initJobs(JobIdx := i)
			THEN
				noOfJobs									:= i;
			ELSE
				EXIT;
			END_IF
		END_FOR

		ModBusCom.DeleteData();
		ModBusCom.noOfJobs									:= noOfJobs;
	
		state												:= 1;
	END_IF

//Read/write slave data is active
1: 
	//Init write data if requesed by master
	IF ModBusCom.writeJobRequested 
	THEN //
		ModBusCom.DeleteData();
		prepareWriteData(currentJobIdx := ModBusCom.currentJobIdx);
		ModBusCom.writeJobRequested 						:= FALSE;
	END_IF
	
	//Evaluation of job result
	IF ModBusCom.Jobs[ModBusCom.currentJobIdx].Valid //Valid is set by master
	THEN	
		Valid 												:= FALSE; //Slave data not valid
		evaluation(CurrentJobIdx := ModBusCom.currentJobIdx);	
				
		countBad 											:= ModBusCom.countBad;
		countGood 											:= ModBusCom.countGood;
		TimeStamp 											:= ModBusCom.Jobs[ModBusCom.currentJobIdx].TimeStamp;
		ModBusCom.Jobs[ModBusCom.currentJobIdx].Valid 		:= FALSE;
		ModBusCom.DeleteData();                                 
		Valid 												:= TRUE; //Slave data valid
		run													:= TRUE;
	ELSE
		run													:= FALSE;
	END_IF
	
	state													:= SEL(Enable, 0, state);
	ModBusCom.Enable										:= Enable;	
END_CASE
END_METHOD

END_FUNCTION_BLOCK

// ---- POUs/ControllerTools/AverageFilter.TcPOU
//LREAL average filter
FUNCTION_BLOCK AverageFilter
VAR_INPUT	
	IN														: LREAL;		// Adds value for average calculation
END_VAR
VAR_OUTPUT
	Q														: LREAL:=0.0;	// Result of average calculation
	Valid													: BOOL:=FALSE;	// Is TRUE once a value is inserted
END_VAR         											
VAR             											
	Total													: LREAL:=0.0;
	Count													: LREAL:=0;
END_VAR

Insert(IN);

METHOD PUBLIC clear : booL; //Return value = TRUE if execution finished
VAR_INPUT
END_VAR
Q:=Total	:=0.0;
Valid		:=FALSE;
Count		:=0.0;
Clear		:= TRUE;
END_METHOD

METHOD PUBLIC insert : LREAL //Result = actual average value
VAR_INPUT
	Value								:	LREAL ;
END_VAR
Total		:=Total+Value;
Count		:=Count+1.0;
Q			:=Total/Count;
Valid		:=TRUE;
Insert 		:= Q;
END_METHOD

END_FUNCTION_BLOCK

// ---- POUs/EventLogger/getEventClassText.TcPOU
//Returns event class in english and upper case letters 
FUNCTION getEventClassText : STRING(12)
VAR_INPUT
	TcEventClass													: E_TcEventClass;
END_VAR
VAR
END_VAR

CASE TcEventClass OF
TC2_SYSTEM.TCEVENTCLASS_NONE		: GetEventClassText 	:= 'NONE';	
TC2_SYSTEM.TCEVENTCLASS_MESSAGE		: GetEventClassText 	:= 'MESSAGE';	
TC2_SYSTEM.TCEVENTCLASS_HINT		: GetEventClassText 	:= 'HINT';	
TC2_SYSTEM.TCEVENTCLASS_STATEINFO	: GetEventClassText 	:= 'STATEINFO';	
TC2_SYSTEM.TCEVENTCLASS_INSTRUCTION	: GetEventClassText 	:= 'INSTRUCTION';			 										
TC2_SYSTEM.TCEVENTCLASS_WARNING		: GetEventClassText 	:= 'WARNING';	
TC2_SYSTEM.TCEVENTCLASS_MAINTENANCE	: GetEventClassText 	:= 'MAINTENANCE';		 														
TC2_SYSTEM.TCEVENTCLASS_ALARM		: GetEventClassText 	:= 'ALARM';	
TC2_SYSTEM.TCEVENTCLASS_PARAMERROR	: GetEventClassText 	:= 'PARAMERROR';		
ELSE
	GetEventClassText										:= 'UNKNOWN';
END_CASE

END_FUNCTION

// ---- POUs/EventLogger/TriggerEvents/EventHandlingGrpCustomized.TcPOU
{attribute 'no_check'}
//Event group with single source id - for a convenient control of <MAX_EVENTS>
//Each single event handling FB is accessible, so that signal flag, information text and alarm class could be used
FUNCTION_BLOCK EventHandlingGrpCustomized
VAR_OUTPUT CONSTANT
	MIN_EVENT												:	INT := 1; 
	MAX_EVENT												:	INT := PARAM.EVENT_HANDLING_CONFIG.GRP_CUSTOMISED_MAX_EVENT; //Start index no of events - see library parameter to customize parameter
END_VAR                                                 	
VAR_INPUT                                               	
	ConfirmTrig												:	BOOL := FALSE; //Acknowledge event
	SourceId												: 	UDINT := 0; //Source id for all events of this group
	no														:	ARRAY [MIN_EVENT..MAX_EVENT] OF EventHandling; //Array of single event handling FBs 
	Disable													:	BOOL := FALSE; //Disable all events 
	AutoConfirm												:	BOOL := FALSE; //All events will be acknowledged if flag is gone *)
	SetClass												:	E_TcEventClass := TC2_SYSTEM.TCEVENTCLASS_ALARM;// if set class is <> ALARM -> all events set to this Eventclass
	MsgOffset												:	INT := 0; //Offset to change default message id to MIN_EVENT to MsgOffset
END_VAR                                                 	
VAR_OUTPUT                                              	
{attribute 'displaymode':='binary'}
	Status													:	DWORD; (*	.0 - .8 = event of <class id> is active / .15 confirm required / .16 = Level 0 , .17 = Level 1 , .18 = Level 2, ..........
																			TCEVENTCLASS_NONE			:=0,	(* No class *)
																			TCEVENTCLASS_MAINTENANCE	:=1,	(* Maintenance hint *)
																			TCEVENTCLASS_MESSAGE		:=2,	(* Message *)
																			TCEVENTCLASS_HINT			:=3,	(* Hint *)
																			TCEVENTCLASS_STATEINFO		:=4,	(* State information *)
																			TCEVENTCLASS_INSTRUCTION	:=5,	(* Instruction *)
																			TCEVENTCLASS_WARNING		:=6,	(* Warning *)
																			TCEVENTCLASS_ALARM			:=7,	(* Alarm *)
																			TCEVENTCLASS_PARAMERROR		:=8		(* Parameter error *)  *)
	NoOfActiveEvents										:	INT;
END_VAR                                                 	
VAR                                                     	
	_Mem													:	BYTE;
	Disabled												:	BOOL;
	i 														:	INT;
END_VAR

(* EventHandlingGrp			V4.1	*)
(************************************)

(* status ***************************)
Status  													:= 0;
NoOfActiveEvents											:= 0;

IF(Disable OR SourceId = 0)AND Disabled
THEN
	RETURN;
ELSE
	Disabled												:= Disable OR SourceId = 0;
	
	FOR i := MIN_EVENT TO MAX_EVENT 
	DO
		(* Init Default Class *)
		IF SetClass <> TC2_SYSTEM.TCEVENTCLASS_ALARM
			AND NOT _Mem.7
		THEN
			no[i].eClass										:= SetClass;
			_Mem.7											:= i = MAX_EVENT;
		END_IF                                  			
		                                        			
		IF Disable OR SourceId = 0              			
		THEN                                    			
			no[i].Flag 										:= FALSE;
			no[i].ConfirmTrig 										:= no[i].State <> TCEVENTSTATE_INVALID AND no[i].State <> TCEVENTSTATE_RESETCON;
		ELSIF ConfirmTrig                             			
		THEN                                    	
			no[i].ConfirmTrig 								:= TRUE;
			_Mem.0 											:= ConfirmTrig;
                                                			
		ELSIF _Mem.0                            			
		THEN                                    			
			no[i].ConfirmTrig 								:= FALSE;
			_Mem.0 											:= i <> MAX_EVENT;

		ELSIF AutoConfirm
		THEN
			IF NOT no[i].Flag
				AND no[i].State <> TCEVENTSTATE_INVALID
				AND no[i].State <> TCEVENTSTATE_RESETCON
			THEN
				no[i].ConfirmTrig 							:= TRUE;
			ELSE                                			
				no[i].ConfirmTrig 							:= FALSE;
			END_IF                              			
		END_IF                                  	
                                                	
		(* Mem current Event *)                 	
		IF no[i].State <> TCEVENTSTATE_INVALID OR no[i].Flag 
		THEN
			_Mem.1											:= TRUE;
			(* Call Event *)
			no[i](
				Flag	:= ,
				ConfirmTrig := ,
				MsgId	:= TO_UINT(i + MsgOffset),
				SourceId:= SourceId,
				eClass	:= (* see grp call *),
				Text1	:= (* see grp call *),
				Text2	:= (* see grp call *),
				pText3	:= (* see grp call *),
				State	=> );
		END_IF

		(* Set info flags *)
		IF	no[i].State <> TCEVENTSTATE_INVALID 
		THEN
			NoOfActiveEvents								:= NoOfActiveEvents + 1;
			Status											:= Status OR no[i].Status;
			Disabled										:= FALSE;
		ELSIF _Mem.1
		THEN (* Send one time info event is gone *)
			; 
		END_IF
	END_FOR	
END_IF
(*****************************************************************************************)

METHOD PUBLIC confirm : booL  //Return value = TRUE if execution finished
VAR_INPUT
END_VAR
IF NoOfActiveEvents > 0
THEN
	FOR i := MIN_EVENT TO MAX_EVENT 
	DO
		no[i](ConfirmTrig := TRUE);
	END_FOR
	_Mem.0			:= TRUE;
END_IF

confirm		:= TRUE;
END_METHOD

END_FUNCTION_BLOCK

// ---- POUs/EventLogger/TriggerEvents/EventHandlingConfirmIsReq.TcPOU
{attribute 'no_check'}
//Returns status of "QuitRequired" configuration for corresponding event class (see library Param) 
FUNCTION EventHandlingConfirmIsReq : BOOL
VAR_INPUT
	TcEventClass											:	E_TcEventClass;
END_VAR
VAR
END_VAR

	CASE tcEventClass OF
	Tc2_System.TCEVENTCLASS_NONE:			EventHandlingConfirmIsReq	:= PARAM.EVENT_HANDLING_CONFIG.CLASS_NONE_QUIT_REQUIRED;	
	Tc2_System.TCEVENTCLASS_MAINTENANCE:	EventHandlingConfirmIsReq	:= PARAM.EVENT_HANDLING_CONFIG.CLASS_MAINTENANCE_QUIT_REQUIRED;		
	Tc2_System.TCEVENTCLASS_MESSAGE:		EventHandlingConfirmIsReq	:= PARAM.EVENT_HANDLING_CONFIG.CLASS_MESSAGE_QUIT_REQUIRED;			
	Tc2_System.TCEVENTCLASS_HINT:			EventHandlingConfirmIsReq	:= PARAM.EVENT_HANDLING_CONFIG.CLASS_HINT_QUIT_REQUIRED;	
	Tc2_System.TCEVENTCLASS_STATEINFO:		EventHandlingConfirmIsReq	:= PARAM.EVENT_HANDLING_CONFIG.CLASS_STATEINFO_QUIT_REQUIRED;	
	Tc2_System.TCEVENTCLASS_INSTRUCTION:	EventHandlingConfirmIsReq	:= PARAM.EVENT_HANDLING_CONFIG.CLASS_INSTRUCTION_QUIT_REQUIRED;	
	Tc2_System.TCEVENTCLASS_WARNING:		EventHandlingConfirmIsReq	:= PARAM.EVENT_HANDLING_CONFIG.CLASS_WARNING_QUIT_REQUIRED;	
	Tc2_System.TCEVENTCLASS_ALARM:			EventHandlingConfirmIsReq	:= PARAM.EVENT_HANDLING_CONFIG.CLASS_ALARM_QUIT_REQUIRED;	
	Tc2_System.TCEVENTCLASS_PARAMERROR:		EventHandlingConfirmIsReq	:= PARAM.EVENT_HANDLING_CONFIG.CLASS_PARAMERROR_QUIT_REQUIRED;		
	ELSE                                                    
		EventHandlingConfirmIsReq										:= PARAM.EVENT_HANDLING_CONFIG.CLASS_ALARM_QUIT_REQUIRED;
	END_CASE

END_FUNCTION

// ---- POUs/Fieldbus/EtherCAT/_Components/EcMasterSupervisor.TcPOU
{attribute 'no_check'}
// Set state of EtherCAT Master(ReqState <> 0) or read state and frame statistic 
// The FB will automatically perform a device reset if the requested state cannot be reached within the TIMEOUT_SET_STATE period
// In addition via options is possible to clear the frame statistic while set or read the Master state
FUNCTION_BLOCK EcMasterSupervisor EXTENDS FbBase
VAR CONSTANT
	TIMEOUT_SET_STATE										:	TIME := T#15S;
END_VAR
VAR_OUTPUT CONSTANT
{attribute 'displaymode':='binary'}
	OPTION_CLEAR_CRC_ERROR_COUNTER							:	BYTE := 2#0000_0001; //delete the CRC error counters of all EtherCAT slaves
{attribute 'displaymode':='binary'}
	OPTION_CLEAR_LOST_FRAMES_COUNTER						:	BYTE := 2#0000_0010; //delete the CRC error counters of all EtherCAT slaves.
{attribute 'displaymode':='binary'}	
	OPTION_CLEAR_TXRX_ERROR_COUNTER							:	BYTE := 2#0000_0100; //delete the error counters of the miniport driver of the network card
{attribute 'displaymode':='binary'}	
	OPTION_FORCE_DEVICE_RESET								:	BYTE := 2#1000_0000; //Force to execute a device reset prior to set state
END_VAR
VAR_INPUT
	AmsNetId												:	T_AmsNetId;	
	DevId													:	WORD;		//Id of mentioned device
{attribute 'displaymode':='binary'}
	Options													:	BYTE := 0; //Select	which error counter should be deleted 
{attribute 'displaymode':='hex'}
	ReqState												:	WORD := 0; (* 	Requested EtherCAT state 
																				EC_DEVICE_STATE_INIT		:BYTE 	:=16#01;
																				EC_DEVICE_STATE_PREOP		:BYTE 	:=16#02;
																				EC_DEVICE_STATE_BOOTSTRAP	:BYTE 	:=16#03;
																				EC_DEVICE_STATE_SAFEOP		:BYTE 	:=16#04;
																				EC_DEVICE_STATE_OP			:BYTE 	:=16#08; *)

END_VAR                     							
VAR_OUTPUT                  										
	ReqStateOK												:	BOOL;	//Requested EtherCAT state OK
{attribute 'displaymode':='hex'}
	CurrState												:	WORD;	//Shows current EtherCAT state
	StateText												:	STRING;	//EtherCAT State as text
	DevResetDone											:	BOOL;	//Device was reseted
//Frames statistic
    LostFrames 												: 	UDINT; //Current number of lost or invalid cyclic frames
    FramesPerSecond 										: 	LREAL; //Current number of cyclic frames per second
    LostQueuedFrames 										: 	UDINT; //Current number of lost or invalid queued (acyclic) frames
    QueuedFramesPerSecond 									: 	LREAL; //Returns the current number of queued (acyclic) frames per second
	
	ErrorText												:	STRING;
END_VAR                     								
VAR                         								
	ErrCntreset													:	INT;
	TON_TimeoutSetStatus									:	TON;
	TON_GetStateTrig										:	TON;
	MemReqState												:	WORD;

	SetMasterState											:	FB_EcSetMasterState := (tTimeout := DEFAULT_ADS_TIMEOUT);
	GetMasterState											:	FB_EcGetMasterState := (tTimeout := DEFAULT_ADS_TIMEOUT);
	ReadMasterFrameStatistic								:	FB_EcMasterFrameStatistic:= (tTimeout := DEFAULT_ADS_TIMEOUT);
	FrameStatisticClearCRC									:	FB_EcMasterFrameStatisticClearCRC:= (tTimeout := DEFAULT_ADS_TIMEOUT);
	FrameStatisticClearFrames								:	FB_EcMasterFrameStatisticClearFrames:= (tTimeout := DEFAULT_ADS_TIMEOUT);
	FrameStatisticClearTxRxErr								:	FB_EcMasterFrameStatisticClearTxRxErr:= (tTimeout := DEFAULT_ADS_TIMEOUT);
	IoDevreset												:	IOF_DeviceReset := (TMOUT := DEFAULT_ADS_TIMEOUT);
END_VAR

	(* Read or set (ReqState <> 0) EtherCAT Master State			*)
	(****************************************************************)

(* Process ******************************************************)
	rtExecute(CLK := Execute);

	CASE state OF
	(* Cyclic reading of state ***********************************)
	0:
		Busy 												:= FALSE;
                                        					
		IF rtExecute.Q THEN            					
			Busy 											:= TRUE;
			Done 											:= FALSE;
			Error											:= FALSE;
			ErrorID											:= 0;
			Errortext										:= '';
			DevResetDone									:= FALSE;
			CurrState										:= 0;
			ReqStateOK										:= FALSE;
			StateText										:= '';
			GetMasterState(bExecute := FALSE,sNetId	:= AmsNetId);
			SetMasterState(bExecute := FALSE,sNetId	:= AmsNetId );
			ReadMasterFrameStatistic(bExecute := FALSE,sNetId	:= AmsNetId );
			FrameStatisticClearCRC(bExecute := FALSE,sNetId	:= AmsNetId );
			FrameStatisticClearFrames(bExecute := FALSE,sNetId	:= AmsNetId );
			FrameStatisticClearTxRxErr(bExecute := FALSE,sNetId	:= AmsNetId );
			IoDevReset(RESET := FALSE);
			TON_TimeoutSetStatus(IN := FALSE);

			IF ReqState <> 0 
				AND (ReqState <> CurrState OR ReqState <> MemReqState)
			THEN
				SetMasterState( bExecute	:= TRUE, reqState	:= ReqState);
				MemReqState 								:= ReqState;
				state 										:= SEL(Options.7, 10, 11) ; //Start with reset device
			ELSE
				(* Start Read Status *)
				GetMasterState(bExecute	:= TRUE);
				state 										:= 1;
			END_IF
		ELSIF NOT Execute THEN
			Done 											:= FALSE;
			DevResetDone 									:= FALSE;
			Error											:= FALSE;
			ErrorID											:= 0;
			ErrorText										:= '';
		END_IF                      					

	(* Read state ******************************************)
	1:
		GetMasterState(bExecute := TRUE);
		IF NOT GetMasterState.bBusy
		THEN
			IF GetMasterState.bError THEN
				Busy										:= FALSE;
				Error										:= TRUE;
				ErrorId										:= GetMasterState.nErrId;
				ErrorText									:= CONCAT('FB_EcGetMasterState Id: ',UDINT_TO_STRING(ErrorId));
				state 										:= 0;
			ELSE                
				CurrState									:= GetMasterState.state;
				ReqStateOK									:= CurrState = ReqState OR ReqState = 0;
				StateText									:= F_ConvStateToString(CurrState);							
				state 										:= state + 1;
			END_IF
		END_IF
		
	(* read frame statistic ******************************************)
	2:
		ReadMasterFrameStatistic(bExecute := TRUE);
		IF NOT ReadMasterFrameStatistic.bBusy
		THEN
			IF ReadMasterFrameStatistic.bError THEN
				Busy										:= FALSE;
				Error										:= TRUE;
				ErrorId										:= ReadMasterFrameStatistic.nErrId;
				ErrorText									:= CONCAT('FB_EcMasterFrameStatistic Id: ',UDINT_TO_STRING(ErrorId));
				state 										:= 0;
			ELSE                
				LostFrames 									:= ReadMasterFrameStatistic.nLostFrames;
				FramesPerSecond 							:= ReadMasterFrameStatistic.fFramesPerSecond;
				LostQueuedFrames 							:= ReadMasterFrameStatistic.nLostQueuedFrames;
				QueuedFramesPerSecond 						:= ReadMasterFrameStatistic.fQueuedFramesPerSecond;		
				state 										:= 20;
			END_IF
		END_IF
		
	(* Set state *****************************************)
	10:
		TON_TimeoutSetStatus(IN := TRUE, PT := TIMEOUT_SET_STATE);
		SetMasterState(bExecute := TRUE);
		IF NOT SetMasterState.bBusy
		THEN
			IF SetMasterState.bError AND DevResetDone
			THEN
				Busy										:= FALSE;
				Error										:= TRUE;
				ErrorId										:= SetMasterState.nErrId;
				ErrorText									:= CONCAT('FB_EcSetMasterState Id: ',UDINT_TO_STRING(ErrorId));
				state 										:= 0;
			ELSIF SetMasterState.currState = MemReqState 
			THEN
				CurrState									:= SetMasterState.currState;
				ReqStateOK									:= CurrState = ReqState;
				StateText									:= F_ConvStateToString(CurrState);			
				state 										:= 2;
			ELSIF DevResetDone          					
			THEN     
				Busy										:= FALSE;                   					
				Error										:= TRUE;
				ErrorId										:= E_AdsErr.DEVICE_ABORTED;
				ErrorText									:= 'Device Reset failed - Master state <> ReqState';
				state 										:= 0;
			ELSE //Try to reset master 
				state 										:= state + 1;
			END_IF                      	
            SetMasterState(bExecute := FALSE);                            	
		ELSIF TON_TimeoutSetStatus.Q 
		THEN
			IF NOT DevResetDone 
			THEN (* try to reset master one time  *)
				state 										:= state + 1;
				IoDevReset(RESET := FALSE);
			ELSE
				Busy										:= FALSE;
				ErrCntReset 								:= ErrCntReset +1;
				Error										:= TRUE;
				ErrorId										:= E_AdsErr.DEVICE_TIMEOUT;
				ErrorText									:= CONCAT('FB_EcSetMasterState busy for more then ', TO_STRING(TIMEOUT_SET_STATE));
				state 										:= 0;
			END_IF  
			SetMasterState(bExecute := FALSE);                						
		END_IF

	11:
		TON_TimeoutSetStatus(IN := FALSE);
		state 												:= state + 1;

	(* Reset Device by setting Error State  **********************)
	12:	
		IoDevReset(DEVICEID	:= DevId,RESET	:= TRUE );
		IF NOT IoDevReset.BUSY
		THEN
			IF IoDevReset.ERR THEN
				Busy										:= FALSE;
				Error										:= TRUE;
				ErrorId										:= IoDevReset.ERRID;
				ErrorText									:= CONCAT('IOF_DeviceReset Id: ',UDINT_TO_STRING(ErrorId));
				state 										:= 0;
			ELSE //Tr to                         					
				Error										:= FALSE;
				ErrorId										:= 0;
				ErrorText									:= '';
				DevResetDone 								:= TRUE;
				TON_TimeoutSetStatus(IN := FALSE);
				state 										:= 10;
			END_IF
		ELSE
			;
		END_IF
		
	(* Start to clear frame statistic **********************************)
	20: 
		FrameStatisticClearCRC(bExecute := Options.0);
		IF NOT FrameStatisticClearCRC.bBusy
		THEN
			IF FrameStatisticClearCRC.bError THEN
				Busy										:= FALSE;
				Error										:= TRUE;
				ErrorId										:= FrameStatisticClearCRC.nErrId;
				ErrorText									:= CONCAT('FB_EcMasterFrameStatisticClearCRC Id: ',UDINT_TO_STRING(ErrorId));
				state 										:= 0;
			ELSE                
				state 										:= state + 1;
			END_IF
		END_IF		
	
	21: 
		FrameStatisticClearFrames(bExecute := Options.1);
		IF NOT FrameStatisticClearFrames.bBusy
		THEN
			IF FrameStatisticClearFrames.bError THEN
				Busy										:= FALSE;
				Error										:= TRUE;
				ErrorId										:= FrameStatisticClearFrames.nErrId;
				ErrorText									:= CONCAT('FB_EcMasterFrameStatisticClearFrames Id: ',UDINT_TO_STRING(ErrorId));
				state 										:= 0;
			ELSE                
				state 										:= state + 1;
			END_IF
		END_IF	

	22: 
		FrameStatisticClearTxRxErr(bExecute := Options.2);
		IF NOT FrameStatisticClearTxRxErr.bBusy
		THEN
			IF FrameStatisticClearTxRxErr.bError THEN
				Busy										:= FALSE;
				Error										:= TRUE;
				ErrorId										:= FrameStatisticClearTxRxErr.nErrId;
				ErrorText									:= CONCAT('FB_EcMasterFrameStatisticClearTxRxErr Id: ',UDINT_TO_STRING(ErrorId));
				state 										:= 0;
			ELSE                
				Busy										:= FALSE;
				Done										:= TRUE;
				state 										:= 0;
			END_IF
		END_IF	
		
	ELSE
		;
	END_CASE
                										
(*********************************************************************)

{attribute 'monitoring' := 'call'}
PROPERTY PUBLIC optClearCRCErrorCounter : BOOL
GET
optClearCRCErrorCounter := Options.0;
END_GET
SET
Options.0 := optClearCRCErrorCounter;
END_SET
END_PROPERTY

{attribute 'monitoring' := 'call'}
PROPERTY PUBLIC optClearLostFramesCounter : BOOL
GET
optClearLostFramesCounter := Options.1;
END_GET
SET
Options.1 := optClearLostFramesCounter;
END_SET
END_PROPERTY

{attribute 'monitoring' := 'call'}
PROPERTY PUBLIC optClearTCRXErrCounter : BOOL
GET
optClearTCRXErrCounter := Options.2;
END_GET
SET
Options.2 := optClearTCRXErrCounter;
END_SET
END_PROPERTY

{attribute 'monitoring' := 'call'}
PROPERTY PUBLIC optForceDevReset : BOOL
GET
optForceDevReset := Options.7;
END_GET
SET
Options.7 := optForceDevReset;
END_SET
END_PROPERTY

END_FUNCTION_BLOCK

// ---- POUs/Fieldbus/Profinet/ProfinetControllerIO.TcPOU
{attribute 'no_check'}
//EL6631 Profinet Controller IOs via EtherCAT
FUNCTION_BLOCK ProfinetControllerIO EXTENDS EcSlaveInfoDataExt
VAR_OUTPUT CONSTANT
	MIN_BOX													:	INT := 1;
	MAX_BOX													:	INT := PARAM.PROFINET_CONTROLLER_DEV_IO_MAX_BOX;
END_VAR
VAR_INPUT
	DevCtrl			 								AT %Q*	:	UINT;
	PnIoBoxCtrl										AT %Q*	:	ARRAY[MIN_BOX ..MAX_BOX] OF UINT;
END_VAR
VAR_OUTPUT
//Device parameter
	DevState		 								AT %I*	:	UINT;		//Link to master device state
	PnIoError										AT %I*	:	UINT;		//Link to master IO error
	PnIoDiag										AT %I*	:	UINT;		//Link to master IO Diag 
                         				
	AoeNetId										AT %I*	:	AMSNETID;		//Link to master AoeNetID
//Box states	             	
	PnIoBoxState									AT %I*	:	ARRAY[MIN_BOX ..MAX_BOX] OF UINT; //Link to box state
	PnIoBoxDiag										AT %I*	:	ARRAY[MIN_BOX ..MAX_BOX] OF UINT; //Link to box diag	
END_VAR                     					             	
VAR       
END_VAR

SUPER^();

END_FUNCTION_BLOCK

// ---- POUs/FileHandling/Basic/ReadDirSimple.TcPOU
{attribute 'no_check'}
//List down all files founded in a directory - specified by file type if needed 
FUNCTION_BLOCK ReadDirSimple EXTENDS FbBase
VAR_OUTPUT CONSTANT
	MIN_ENTRYS												:	INT := 1;	
	MAX_ENTRYS												:	INT := PARAM.READ_DIR_SIMPLE_MAX_ENTRYS;	//see library parameter to customize parameter	
	MAX_STRING_LEN											:	INT := PARAM.READ_DIR_SIMPLE_MAX_STRING_LEN;//see library parameter to customize parameter
END_VAR            										  										
VAR_INPUT           										
	AMSNetId												:	T_AmsNetId; //AMS Net Id
	Timeout													:	TIME := DEFAULT_ADS_TIMEOUT; //ADS Timeout Default 3s 
	Path													:	T_MaxString; // \\PC-Name\Folder\ C:\Folder\
	File													:	STRING(MAX_STRING_LEN) := '*.*'; // *.xml / *.txt
END_VAR
VAR_OUTPUT
	NoOfFiles												:	INT; //Number of files found in folder 
	EoE														:	BOOL; //end of enumeration - No more files in folder
	Entry													:	ARRAY[MIN_ENTRYS..MAX_ENTRYS] OF STRING(MAX_STRING_LEN); //List of file names
END_VAR
VAR
(* internal used variables ************************************************************)

(* trigger ****************************************************************************)	

(* function-block instances ***********************************************************)
	EnumFindFileEntry										:	FB_EnumFindFileEntry;
END_VAR


(* Sequence ****************************************)
	rtExecute(CLK := Execute);
	CASE state OF 
	0:	
		Busy												:= FALSE;
		IF NOT Execute
		THEN
			Done											:= FALSE;
			Error											:= FALSE;
			ErrorId											:= 0;
		ELSIF rtExecute.Q
		THEN
			EnumFindFileEntry(bExecute := FALSE, sNetId := AMSNetId, tTimeout := Timeout, sPathName := CONCAT(Path,File));
			Busy											:= TRUE;
			Done											:= FALSE;
			Error											:= FALSE;
			ErrorId											:= 0;
			NoOfFiles										:= 0;
			MEMSET(ADR(Entry),0,SIZEOF(Entry));
			state											:= State + 1;
		END_IF 
	
	1: //read first entry
		EnumFindFileEntry(bExecute := TRUE ,eCmd := eEnumCmd_First );
		state												:= State + 1;

	2: //read entrys
		EnumFindFileEntry(bExecute := TRUE);
		IF NOT EnumFindFileEntry.bBusy
		THEN
			IF NOT EnumFindFileEntry.bError
			THEN
				IF EnumFindFileEntry.bEOE		
				THEN
					Busy									:= FALSE;
					Done									:= TRUE;	
					state									:= 0;
					
				ELSIF NOT EnumFindFileEntry.stFindFile.fileAttributes.bDirectory
				THEN
					NoOfFiles								:= LIMIT(MIN_ENTRYS, NoOfFiles + 1 ,MAX_ENTRYS);
					Entry[NoOfFiles]						:= EnumFindFileEntry.stFindFile.sFileName;
					
					IF EnumFindFileEntry.bEOE
					THEN
						EoE									:= TRUE;
						Busy								:= FALSE;
						Done								:= TRUE;
						state								:= 0;
					ELSIF NoOfFiles >= MAX_ENTRYS
					THEN
						state								:= 3;
					ELSE
						; //Continue with next cycle					
					END_IF		
					
				END_IF
				EnumFindFileEntry(bExecute := FALSE ,eCmd := eEnumCmd_Next);
			ELSE
				Busy										:= FALSE;
				Done										:= FALSE;
				Error										:= TRUE;
				ErrorId										:= EnumFindFileEntry.nErrID;
				state										:= 0;
			END_IF		
		END_IF
		
	3: //End search
		EnumFindFileEntry(bExecute := TRUE ,eCmd := eEnumCmd_Abort);
		IF NOT EnumFindFileEntry.bBusy
		THEN
			Busy											:= FALSE;
			Done											:= NOT EnumFindFileEntry.bError;
			Error											:= NOT Done;
			ErrorId											:= EnumFindFileEntry.nErrID;
			state											:= 0;		
		END_IF
	
	END_CASE

(*************************************************************************)

END_FUNCTION_BLOCK

// ---- POUs/FileHandling/TF6421-XmlServer/XmlReadWrite.TcPOU
{attribute 'no_check'}
//Wrapper for functions of TF6421 XML-Server
//based on TF6421 - required lib: Tc2_XmlDataSvr - see Beckhoff documentation for more information
FUNCTION_BLOCK XmlReadWrite EXTENDS FbBase
VAR_OUTPUT CONSTANT
	FNC_READ												:	INT := 0; //Read data from XML
	FNC_WRITE												:	INT := 1; //Create XML if not exist and wite data into file
END_VAR             										
VAR_INPUT           										
	Fnc														:	INT (FNC_READ..FNC_WRITE) := FNC_READ; //See output constants for possible parameter
	NetId													: 	T_AmsNetId := ''; //Ams Net ID
	Mode													: 	WORD := XMLSRV_ADDMISSING; // XMLSRV_SKIPMISSING or XMLSRV_ADDMISSING;
	pSymAddr												: 	PVOID := 0;	//Pointer to target variable to read or write data 
	SymSize													:	UDINT := 0;	//Size of variable/structure
	FilePath												:	T_MaxString := 'C:\'; // \\PCName\Folder\test.xml
	FileName												:	T_MaxString := 'data.xml'; // \\PCName\Folder\test.xml
	XPath													:	T_MaxString := '/dataentry/data'; // XML tag name/adress to access all or specified data insite the file. Array access->CONCAT('/Datentry/Step[@index="',CONCAT(DINT_TO_STRING(AktStep),'"]')); 										
	Timeout													: 	TIME := T#60S;
END_VAR             										
VAR_OUTPUT          										
END_VAR             	
VAR                 	
(* Local variables ************************************************************)
	MemFnc													:	INT := -1;
	
(* Trigger *****************************************************************)

(* Timer ******************************************************************)

(* Fcuntion blocks ***************************************************************)
	XmlSrvRead 												: 	FB_XmlSrvRead;
	XmlSrvWrite 											: 	FB_XmlSrvWrite;

(* Dummys **********************************************************)

END_VAR

	(* XML Read/Write														V2.0		*)
	(************************************************************************************)

(* Execute ***************************************************************************************)
	rtExecute(CLK := Execute);
	IF rtExecute.Q
		AND MemFnc < 0
	THEN
		MemFnc 												:= SEL(Fnc = FNC_WRITE, FNC_READ , FNC_WRITE) ;
		Busy												:= TRUE;
		Done												:= FALSE;
		Error												:= FALSE;
		ErrorID												:= 0;
	END_IF

(* Call Method ***********************************************************************************)
	CASE MemFnc OF
	FNC_READ:
		Read(
			Execute	:= Execute);
	
	FNC_WRITE:
		Write(			
			Execute	:= Execute);
			
	-1:
		IF NOT Execute
		THEN
			Busy											:= FALSE;
			Done											:= FALSE;
			Error											:= FALSE;
			ErrorID											:= 0;
		END_IF                              				
	ELSE                                    				
		Busy												:= FALSE;
		Done												:= FALSE;
		Error												:= Execute;
		ErrorID												:= E_AdsErr.DEVICE_INVALIDPARM;
	END_CASE

(*************************************************************************************************)

METHOD PUBLIC read : BOOL //Return value = TRUE if busy
//required parameter
//pSymAddr
//SymSize
//FilePath
//XPath
VAR_INPUT
	Execute													:	BOOL;
END_VAR
IF pSymAddr = 0 THEN
	Busy													:= NOT Error;
	Error													:= TRUE;
	ErrorId													:= E_AdsErr.DEVICE_INVALIDPARM;
	Done													:= FALSE;
	MemFnc													:= -1 ;
	RETURN;
END_IF

	IF Execute
	THEN
		Error												:=	FALSE;
		ErrorId												:= 0;
		XmlSrvRead.bExecute 								:= TRUE;
	ELSIF NOT XmlSrvRead.bBusy      						
	THEN                            						
		Error												:=	FALSE;
		ErrorId												:= 0;
		XmlSrvRead.bExecute 								:= FALSE;
                                    						
	END_IF                          						
                                    	
	MemFnc													:= FNC_READ;
	                                						
	THIS^.Execute											:= Execute;
                                    						
	XmlSrvRead(                    	
		sNetId		:= NetId,
		ePath		:= ,(* Default *)
		nMode		:= XMLSRV_SKIPMISSING, 
		pSymAddr	:= pSymAddr,
		cbSymSize	:= SymSize,
		sFilePath	:= CONCAT(FilePath,FileName),
		sXPath		:= XPath,
		bExecute	:=  ,
		tTimeout	:= Timeout,
		bBusy		=> Busy,
		bError		=> ,
		nErrId		=> );

	Done													:= NOT XmlSrvRead.bBusy
																AND NOT XmlSrvRead.bError
																AND XmlSrvRead.bExecute;
                                        				
	IF NOT Busy
	THEN
		IF XmlSrvRead.bExecute
		THEN
			Error											:=	XmlSrvRead.bError;
			ErrorId											:= XmlSrvRead.nErrId;
		END_IF
		IF NOT Execute
		THEN
			MemFnc											:= -1 ;
			XmlSrvRead(bExecute := FALSE);
		END_IF
	END_IF
	
	Read													:= Busy;
END_METHOD

METHOD PUBLIC write : BOOL //Return value = TRUE if busy
//required parameter
//pSymAddr
//SymSize
//FilePath
//XPath
VAR_INPUT
	Execute				:	BOOL;
END_VAR
IF pSymAddr = 0 
THEN
	Busy													:= NOT Error;
	Error													:= TRUE;
	ErrorId													:= E_AdsErr.DEVICE_INVALIDPARM;
	Done													:= FALSE;
	MemFnc													:= -1 ;
	RETURN;
END_IF

	IF Execute
	THEN
		Error												:=	FALSE;
		ErrorId												:= 0;
		XmlSrvWrite.bExecute 								:= TRUE;
	ELSIF NOT XmlSrvWrite.bBusy     						
	THEN                            						
		XmlSrvWrite.bExecute								:= FALSE;
		Error												:=	FALSE;
		ErrorId												:= 0;
	END_IF                          						
                                    						
	MemFnc													:= FNC_WRITE;
	                                						
	THIS^.Execute											:= Execute;
                                    	
	XmlSrvWrite(
		sNetId		:= NetId,
		ePath		:= ,(* Default *)
		nMode		:= Mode,
		pSymAddr	:= pSymAddr,
		cbSymSize	:= SymSize,
		sFilePath	:= CONCAT(FilePath,FileName),
		sXPath		:= XPath,
		bExecute	:= ,
		tTimeout	:= Timeout,
		bBusy		=> Busy,
		bError		=> ,
		nErrId		=> );

	Done													:= NOT XmlSrvWrite.bBusy
																AND NOT XmlSrvWrite.bError
																AND XmlSrvWrite.bExecute;
                                        					
	IF NOT Busy
	THEN
		IF XmlSrvWrite.bExecute
		THEN
			Error											:=	XmlSrvWrite.bError;
			ErrorId											:= XmlSrvWrite.nErrId;
		END_IF
		IF NOT Execute
		THEN
			MemFnc											:= -1;
			XmlSrvWrite(bExecute := FALSE);
		END_IF
	END_IF

	Write													:= Busy;
END_METHOD

END_FUNCTION_BLOCK

// ---- POUs/IO/BlowOffSensors.TcPOU
{attribute 'no_check'}
//FB generates a pulse "Pulse" time based signal on every bit at Q (DWORD) for a certain lenght
//The sequecne will starts based on the seletcted time of interval if Enable is TRUE
//The FB can be used to activate air blow valves on by one to clean sensors in a dusty environment
FUNCTION_BLOCK BlowOffSensors
VAR_INPUT
	Enable													:	BOOL;			//FB will be processed as long as enable is TRUE
	StartManual												:	BOOL;			//starts FB without interval
	Interval												:	TIME := T#60M; 	//Blow of autostart interval
	Lenght													:	TIME := T#4S; 	//Duration of pulsing
	Pulse													:	TIME := T#500MS; //On/Off pulse duration
END_VAR                 									
VAR_OUTPUT              									
	Aktiv													:	BOOL;			//Busy is TRUE at the rising edge of Enable and stays TRUE as long as the FB is performing any action.  
{attribute 'displaymode':='binary'}    
	Q														:	DWORD := 0;		//Each bit will be set and reset based on the settings one by one 
END_VAR                 									
VAR                     									
	state													:	INT := 0;
	i														:	SINT ;
	TON_Interval											:	TON;
	TON_Lenght		 										: 	TON;
	TOF_Pulse	 											:	TOF;
END_VAR

(* Abblastaktgenerator					*)
(***************************************)

(* Intervalzeit ***********************************************************************)
IF Enable 
THEN
	CASE state OF
	0:
		TON_Interval(IN := FALSE);
		state 												:= 10;
		i 													:= -1;

	1:
		Aktiv := FALSE;
		TON_Interval(IN := Interval <> T#0MS , PT := Interval);
		IF TON_Interval.Q
			OR StartManual
		THEN
			TON_Interval(IN := FALSE);
			
			state 											:= 10;
			Aktiv 											:= TRUE;
			i 												:= -1;
		END_IF

	10:
		i := i + 1;
		IF i > 31 THEN
			state 											:= 1;
		ELSE
			TON_Lenght(IN := FALSE);
			TOF_Pulse(IN := FALSE);
			
			Q		 										:= 0;
			state 											:= 11;
		END_IF                  							

	11:
		TON_Lenght(IN := TRUE, PT := Lenght);

		IF 	TON_Lenght.Q
			AND Q = 0
		THEN
			state 											:= 10;
		ELSE
			IF 	NOT TOF_Pulse.Q 
				AND Q <> 0 
			THEN
				TOF_Pulse(IN:=TRUE  , PT:= Pulse);
				Q		 									:= 0;
			ELSIF NOT TOF_Pulse.Q 
				AND Q = 0 
			THEN
				TOF_Pulse(IN:= TRUE , PT:= Pulse) ;
				Q		 									:= SETBIT32(Q,i);
			END_IF
			(* Work Timer *)
			TOF_Pulse(IN:=FALSE);
		END_IF

	END_CASE
ELSE
	Aktiv 													:= FALSE;
	state 													:= 0;
	Q														:= 0;
END_IF

(**********************************************************************************************************)

END_FUNCTION_BLOCK

// ---- POUs/TimeHelper/Pulse.TcPOU
{attribute 'no_check'}
//Generates a pulse signal 
FUNCTION_BLOCK Pulse
VAR_INPUT
	IN														: BOOL; //Start pulse generator
	PT_ON													: TIME; //Time pulse on	
	PT_OFF													: TIME; //Time pulse off 
END_VAR             										
VAR_OUTPUT          										
	Q														: BOOL; 
	RT														: BOOL; 
	FT														: BOOL;
END_VAR             										
VAR                 	
	TON_PULSE												: TON;
END_VAR

	(* Pulse generator																*)
	(********************************************************************************)

(* Reset flag *)
RT := FT													:= FALSE;
(* logic *)
IF 	Q AND(TON_PULSE.Q OR NOT IN)
THEN
	TON_PULSE(IN:=FALSE  , PT:= PT_OFF);
	FT 														:= Q;
	Q 														:= FALSE;
ELSIF NOT Q AND TON_PULSE.Q
	OR_ELSE In AND NOT TON_PULSE.IN 
THEN
	RT 														:= NOT Q;
	TON_PULSE(IN:= FALSE , PT:= PT_ON) ;
	Q 														:= TRUE;
END_IF

//Run timer
TON_PULSE(IN:=IN);

(***********************************************************************************************************************)

END_FUNCTION_BLOCK

// ---- POUs/IO/Cylinder/CylinderExt.TcPOU
{attribute 'no_check'}
//Cylinder with runtime status, extended from FB Cylinder
FUNCTION_BLOCK CylinderExt EXTENDS Cylinder 
VAR_OUTPUT CONSTANT
END_VAR
VAR_INPUT  

END_VAR                                     			
VAR_OUTPUT     			
	RuntimeWP												:	TIME;
	RuntimeBP												:	TIME;
END_VAR
VAR
END_VAR

	(* Cylinder	with runtime status 												*)
	(********************************************************************************)

(* Call super ********************************************************)
	SUPER^();
	
(*********************************************************************)

METHOD PROTECTED _runtimeChk : BOOL
VAR_INPUT
END_VAR
VAR
	memRtBP												:	TIME;
	memRtWP												:	TIME;
END_VAR
(* Record current runtime **********************************************)
	memRtBP													:= tonErrBasePos.ET;
	memRtWP													:= TonErrWorkPos.ET;
	
(* Call time *********************************************************)
	SUPER^._runtimeChk();
	
(* Record last runtime *********************************************)
	IF memRtWP > T#0MS AND NOT tonErrWorkPos.IN AND NOT tonErrWorkPos.Q
	THEN
		RuntimeWP											:= memRtWP;
	END_IF
	
	IF memRtBP > T#0MS AND NOT tonErrBasePos.IN AND NOT tonErrBasePos.Q
	THEN
		RuntimeBP											:= memRtBP;
	END_IF
					
(*********************************************************************)
	_runtimeChk												:= TRUE;

(**********************************************************************)
END_METHOD

END_FUNCTION_BLOCK

// ---- POUs/IO/Drives/AxDriveBase.TcPOU
{attribute 'no_check'}
FUNCTION_BLOCK AxDriveBase EXTENDS EcSlaveInfoDataExt IMPLEMENTS I_AxDriveBase
VAR CONSTANT         	
END_VAR  
VAR_INPUT
	rAxis													:	REFERENCE TO AXIS_REF := 0; //Reference to NC-Axis REF
END_VAR                     					
VAR_IN_OUT                  					
END_VAR                     					
VAR_OUTPUT                  					
	Fault													:	BOOL; (* Drive Error *)
	SwitchedOn												:	BOOL; (* Drive enabled *)
	Ready													:	BOOL; (* Drive Ready *)
{attribute 'displaymode':='binary'}    
	Statusword										AT %I* 	:	UINT; //Link to the drive status word after linking the NC
	Channel											AT %I*	:	USINT;
END_VAR                     					                   					
VAR                         				

END_VAR
VAR

(* Cache *********************************************************************)
	State													:	INT; //State machine 

(* Timer ********************************************************************************)

(* Trigger ******************************************************************************)

(* Instance ****************************************************************************)
	
(* Dummy Speicher **********************************************************)
END_VAR

	(* Drive base information															*)
	(************************************************************************************)
	
	SUPER^();

PROPERTY PUBLIC rAxDrive : REFERENCE TO AxDriveBase
GET
rAxDrive REF= This^;
END_GET
END_PROPERTY

PROPERTY Public rInfoData : reference to EcSlaveInfoData
GET
rInfoData REF= THis^;
END_GET
END_PROPERTY

END_FUNCTION_BLOCK

// ---- POUs/IO/Drives/CoE/CiA_DS402Controlword.TcPOU
FUNCTION_BLOCK CiA_DS402Controlword
VAR_INPUT
	SwitchOn 				: BOOL;	// BIT 0 
	EnableVoltage 			: BOOL := TRUE; // Bit 1  
	QuickStopOK 			: BOOL := TRUE; // Bit 2 inverse signal / TRUE = RUN -
	EnableOperation 		: BOOL; // Bit 3 
//	Operation mode specific Bit 4 	: BOOL; // Bit 4
//	Operation mode specific Bit 5 	: BOOL; // Bit 5
//	Operation mode specific Bit 6 	: BOOL; // Bit 6
	FaultReset 				: BOOL; // Bit 7 
	Halt 					: BOOL; // Bit 8 - Pauses the drive in all modes
//	Operation mode specific Bit 9 	: BOOL; // Bit 9 - 
//	Reserved Bit 10 	: BOOL; // Bit 10
//	Manufacturere specific Bit 11 	: BOOL; // Bit 11
//	Manufacturere specific Bit 12 	: BOOL; // Bit 12
//	Manufacturere specific Bit 13 	: BOOL; // Bit 13
//	Manufacturere specific Bit 14 	: BOOL; // Bit 14
//	Manufacturere specific Bit 15 	: BOOL; // Bit 15	
END_VAR
VAR_OUTPUT
	Cmd						:	eCiA_DS402_CONTROL_CMD;
END_VAR
VAR
END_VAR

;

METHOD PUBLIC createControlword : BOOL
VAR_INPUT
	StatusState												: 	eCiA_DS402_STATUS_STATE;
END_VAR
VAR_IN_OUT
	Controlword												:	UINT;
END_VAR
(* work local state machine for control ****************************************************)
	CASE StatusState OF
	eCiA_DS402_STATUS_STATE.NOT_READY_TO_SWITCH_ON:
		Controlword.0										:= FALSE;
		Controlword.1										:= FALSE;
		Controlword.2										:= FALSE;
		Controlword.3										:= FALSE;
		Cmd													:= eCiA_DS402_CONTROL_CMD.DISABLE_VOLTAGE;
		
	eCiA_DS402_STATUS_STATE.SWITCH_ON_DISABLED:
		IF EnableVoltage
		THEN //back to "not ready to switch on"
			Controlword.0									:= FALSE;
			Controlword.1									:= TRUE;
			Controlword.2									:= TRUE;
			Controlword.3									:= FALSE;
			Cmd												:= eCiA_DS402_CONTROL_CMD.SHUTDOWN;
		ELSE //To "Ready to switch on"
			Controlword.0									:= FALSE;
			Controlword.1									:= FALSE;
			Controlword.2									:= FALSE;
			Controlword.3									:= FALSE;
			Cmd												:= eCiA_DS402_CONTROL_CMD.DISABLE_VOLTAGE;
		END_IF
		
	eCiA_DS402_STATUS_STATE.READY_TO_SWITCH_ON:
		IF NOT EnableVoltage
		THEN //Back to switched on disabled
			Controlword.0									:= FALSE;
			Controlword.1									:= FALSE;
			Controlword.2									:= FALSE;
			Controlword.3									:= FALSE;
			Cmd												:= eCiA_DS402_CONTROL_CMD.DISABLE_VOLTAGE;
		ELSIF SwitchOn
		THEN //To switched on
			Controlword.0									:= TRUE;
			Controlword.1									:= TRUE;
			Controlword.2									:= QuickStopOK;
			Controlword.3									:= FALSE;
			Cmd												:= eCiA_DS402_CONTROL_CMD.SWITCH_ON;	
		ELSE
			Controlword.0									:= FALSE;
			Controlword.1									:= TRUE;
			Controlword.2									:= QuickStopOK;
			Controlword.3									:= FALSE;
			Cmd												:= eCiA_DS402_CONTROL_CMD.SHUTDOWN;			
		END_IF	
		
